	SR_TempDeviationToHighB[5](SET1:=mxAutoMode AND
((BottomMoldB.HeatingZone[5].FB_Temperature.EngTempOut > TopMoldB.HeatingZone[5].FB_Temperature.EngTempOut + 40.0)  OR 
( BottomMoldB.HeatingZone[5].FB_Temperature.EngTempOut < TopMoldB.HeatingZone[5].FB_Temperature.EngTempOut - 40.0)), RESET:=mxReset, Q1=>Errors.TempDeviationToHighB[5]);

	SR_TempDeviationToHighB[6](SET1:=mxAutoMode AND
((BottomMoldB.HeatingZone[6].FB_Temperature.EngTempOut > TopMoldB.HeatingZone[6].FB_Temperature.EngTempOut + 40.0)  OR 
( BottomMoldB.HeatingZone[6].FB_Temperature.EngTempOut < TopMoldB.HeatingZone[6].FB_Temperature.EngTempOut - 40.0)), RESET:=mxReset, Q1=>Errors.TempDeviationToHighB[6]);


(*Red hot safetyrule Regading heating Transfermold may not move down when bottommold A or B isn't hot enough*)
ASideNotWarm :=  ((BottomMoldA.HeatingZone[1].FB_Temperature.EngTempOut < MachParameters.MinTempAlowTransferToBot) AND MachParameters.BottomMoldA.HeatingZone[1].mxZoneActive) OR
				 ((BottomMoldA.HeatingZone[2].FB_Temperature.EngTempOut < MachParameters.MinTempAlowTransferToBot) AND MachParameters.BottomMoldA.HeatingZone[2].mxZoneActive) OR
				 ((BottomMoldA.HeatingZone[3].FB_Temperature.EngTempOut < MachParameters.MinTempAlowTransferToBot) AND MachParameters.BottomMoldA.HeatingZone[3].mxZoneActive) OR
				 ((BottomMoldA.HeatingZone[4].FB_Temperature.EngTempOut < MachParameters.MinTempAlowTransferToBot) AND MachParameters.BottomMoldA.HeatingZone[4].mxZoneActive) OR
				 ((BottomMoldA.HeatingZone[5].FB_Temperature.EngTempOut < MachParameters.MinTempAlowTransferToBot) AND MachParameters.BottomMoldA.HeatingZone[5].mxZoneActive) OR
				 ((BottomMoldA.HeatingZone[6].FB_Temperature.EngTempOut < MachParameters.MinTempAlowTransferToBot) AND MachParameters.BottomMoldA.HeatingZone[6].mxZoneActive);
		
BSideNotWarm :=  ((BottomMoldB.HeatingZone[1].FB_Temperature.EngTempOut < MachParameters.MinTempAlowTransferToBot) AND MachParameters.BottomMoldB.HeatingZone[1].mxZoneActive) OR
				 ((BottomMoldB.HeatingZone[2].FB_Temperature.EngTempOut < MachParameters.MinTempAlowTransferToBot) AND MachParameters.BottomMoldB.HeatingZone[2].mxZoneActive) OR
				 ((BottomMoldB.HeatingZone[3].FB_Temperature.EngTempOut < MachParameters.MinTempAlowTransferToBot) AND MachParameters.BottomMoldB.HeatingZone[3].mxZoneActive) OR
				 ((BottomMoldB.HeatingZone[4].FB_Temperature.EngTempOut < MachParameters.MinTempAlowTransferToBot) AND MachParameters.BottomMoldB.HeatingZone[4].mxZoneActive) OR
				 ((BottomMoldB.HeatingZone[5].FB_Temperature.EngTempOut < MachParameters.MinTempAlowTransferToBot) AND MachParameters.BottomMoldB.HeatingZone[5].mxZoneActive) OR
				 ((BottomMoldB.HeatingZone[6].FB_Temperature.EngTempOut < MachParameters.MinTempAlowTransferToBot) AND MachParameters.BottomMoldB.HeatingZone[6].mxZoneActive);
				
// FMEA (140 degree?)
SR_BotMoldAToCoolForTrMDown(SET1:=NOT mxCommisioningMode AND (BottomMoldA.mxCilIsIn AND ASideNotWarm AND TransferMold.mxCilIsMovingOut), Reset:=mxReset, Q1=>Errors.RH_BotMoldAToCoolForTrMDown);

SR_BotMoldBToCoolForTrMDown(Set1:= NOT mxCommisioningMode AND (BottomMoldB.mxCilIsIn AND BSideNotWarm AND TransferMold.mxCilIsMovingOut), reset:=mxReset, Q1=>Errors.RH_BotMoldBToCoolForTrMDown);
END_ACTION

ACTION Init:
(*StateChange (Transition)  Signalgeneration*)
mxInitTransitionState:=(miInitState<>miInitOldstate);
(*State text*)
sInitStateText:=sInitStateTextDef[miInitState];
(*Timeout Watchdog for Statemachine*)
mxInitTimeoutEnable:=NOT (miInitState=0)  AND NOT mxReset;

InitTimeout(IN:=mxInitTimeoutEnable  , PT:=tInitStateTimeouts[miInitState] );
InitTimeOutUpFlank(CLK:=InitTimeout.Q );
miInitOldstate:=miInitState;

(*Set Errorbit when Raising edge of Timeout has been detected*)
IF InitTimeOutUpFlank.Q THEN
	exInitTimeOut:=TRUE; 			(* 1 Timeout for the whole programcycle *)
END_IF

(*Function to reset the Statemachine*)
IF mxResetInitState THEN
	mxResetInitState:=FALSE;
	miInitState:=0;
	miInitOldstate:=miInitState;
	mxInitTransitionState:=FALSE;

	mxStartInit:= FALSE;
	mxStopInit:= FALSE;
	
	TopMoldA.mxResetInitState:= TRUE;
	TopMoldB.mxResetInitState:= TRUE;
	BottomMoldA.mxResetInitState:= TRUE;
	BottomMoldB.mxResetInitState:= TRUE;
	TransferMold.mxResetInitState:= TRUE;
	ProductForming.mxResetInitState:= TRUE;
	
END_IF

(*Definition State has Error*)
mxInitHasError:=FALSE;

(*Init State's*)
CASE miInitState OF
	0:
		IF mxStartInit THEN
			mxStartInit:= FALSE;
			mxInitialized:= FALSE;
			
			TransferMold.M_StartInit();
			ProductForming.M_StartInit();
			
			//HydraulicsMain.HydraulicPump.M_Start();
		
			miInitState:= 2;
		END_IF

	(* Init Transfermold / Product Forming*)
	2:
		IF mxStopInit THEN
			mxStopInit:= FALSE;
			
			miInitState:= 10;
		ELSIF TransferMold.mxInitialized AND ProductForming.mxInitialized THEN 
			IF MachParameters.EnableEamcSideA THEN
				TopMoldA.M_StartInit(); 

				miInitState:= 3;
			ELSIF MachParameters.EnableEamcSideB THEN
				TopMoldB.M_StartInit();

				miInitState:= 5; 
			END_IF
		END_IF

	(* Init topMold A *)
	3:
		IF mxStopInit THEN
			mxStopInit:= FALSE;
			
			miInitState:= 10;
		ELSIF TopMoldA.mxInitialized THEN
			BottomMoldA.M_StartInit();

			miInitState:= 4;
		END_IF

	(* Init BottomMold A *)	
	4:
		IF mxStopInit THEN
			mxStopInit:= FALSE;
			
			miInitState:= 10;
		ELSIF BottomMoldA.mxInitialized THEN
			IF MachParameters.EnableEamcSideB THEN
				TopMoldB.M_StartInit();

				miInitState:= 5; 
			ELSE
				//HydraulicsMain.M_SartInit();
				
				miInitState:= 7;
			END_IF
		END_IF

	(* Init topMold B *)
	5:
		IF mxStopInit THEN
			mxStopInit:= FALSE;
			
			miInitState:= 10;
		ELSIF TopMoldB.mxInitialized THEN
			BottomMoldB.M_StartInit();

			miInitState:= 6;
		END_IF

	(* Init BottomMold B *)	
	6:
		IF mxStopInit THEN
			mxStopInit:= FALSE;
			
			miInitState:= 10;
		ELSIF BottomMoldB.mxInitialized THEN
			//HydraulicsMain.M_SartInit();

			miInitState:= 7;
		END_IF

	(* Initialized *)
	7:
		mxInitialized:= TRUE;
		miInitState:= 0;
		
		//HydraulicsMain.HydraulicPump.M_Stop();
	(* Stop init *)
	10:
		mxInitialized:= FALSE;

		//HydraulicsMain.HydraulicPump.M_Stop();
		
		IF TopMoldA.mxInitBusy THEN TopMoldA.M_StopInit(); END_IF
		IF TopMoldB.mxInitBusy THEN TopMoldB.M_StopInit(); END_IF
		IF BottomMoldA.mxInitBusy THEN BottomMoldA.M_StopInit(); END_IF
		IF BottomMoldB.mxInitBusy THEN BottomMoldB.M_StopInit(); END_IF
		IF TransferMold.mxInitBusy THEN TransferMold.M_StopInit(); END_IF
		IF ProductForming.mxInitBusy THEN ProductForming.M_StopInit(); END_IF
		IF HydraulicsMain.mxInitbusy THEN HydraulicsMain.M_StopInit(); END_IF		

		miInitState:=11;
		
	(* Stop Init *)
	11:
		IF NOT TopMoldA.mxInitBusy AND NOT TopMoldB.mxInitBusy AND NOT BottomMoldA.mxInitBusy AND NOT BottomMoldB.mxInitBusy AND NOT TransferMold.mxInitBusy 
			AND NOT ProductForming.mxInitBusy AND NOT HydraulicsMain.mxInitbusy THEN	

			
			
			miInitState:= 0;
		END_IF
END_CASE

mxInitBusy:= miInitState<>0;
END_ACTION

METHOD M_StartCycle

IF (NOT mxCycleBusy AND mxInitialized) OR (mxInPause AND mxInitialized) THEN
	mxInPause:= FALSE;
	mxStartCycle:= TRUE;	
END_IF
END_METHOD

METHOD M_StartHydraulics : BOOL
HydraulicsMain.M_StartCycle();
END_METHOD

METHOD M_StartInit

IF NOT mxInitBusy THEN 
	mxStartInit:= TRUE; 
END_IF
END_METHOD

METHOD M_StopCycle

IF mxCycleBusy THEN
	mxStopCycle:= TRUE;	
	mxInPause:=TRUE;
END_IF
END_METHOD

METHOD M_StopCycleEmpty

IF mxCycleBusy THEN 
	mxStopCycleEmpty:= TRUE; 
END_IF
END_METHOD

METHOD M_StopDirect

IF mxCycleBusy THEN
	mxStopDirect:= TRUE;	
END_IF
END_METHOD

METHOD M_StopHydraulics
HydraulicsMain.M_StopCycleEmpty();
END_METHOD

METHOD M_StopInit

IF mxInitBusy THEN 
	mxStopInit:= TRUE; 
END_IF
END_METHOD

ACTION Objects:

TopMoldA(
	mxReset:= mxReset,
	mxEmergency:= mxEmergency[8],
	mxDoorsOpened:= mxEmergency[2] OR mxEmergency[3],
	mxAutoMode:= mxAutoMode,
	mxEnableHeating:= mxEnableHeating,	
	mxTakeOutIsMovingUp:= BottomMoldA.mxTakeoutIsMovingUp, 
	ActualPositionTransfermold:=Transfermold.ActualPosition,	
	RHSR_Blocked:= Errors.RH_ToMoldAIsMovingBoMoldANotInPos,
	MachParameters:= MachParameters.TopMoldA,
	ProdParameters:= ProdParameters.TopMoldA,
	Errors=> Errors.TopMoldA);

TopMoldB(
	mxReset:= mxReset,
	mxEmergency:= mxEmergency[8],
	mxDoorsOpened:=mxEmergency[3] OR mxEmergency[4],
	mxAutoMode:= mxAutoMode,
	mxEnableHeating:= mxEnableHeating,		
	mxTakeOutIsMovingUp:= BottomMoldB.mxTakeoutIsMovingUp, 
	ActualPositionTransfermold:=Transfermold.ActualPosition,
	RHSR_Blocked := Errors.RH_ToMoldBIsMovingBoMoldBNotInPos,
	MachParameters:= MachParameters.TopMoldB,
	ProdParameters:= ProdParameters.TopMoldB,
	Errors=> Errors.TopMoldB);
	
BottomMoldA(
	mxReset:= mxReset,
	mxEmergency:=mxEmergency[8],
	mxDoorsOpened:= mxEmergency[2] OR mxEmergency[3],
	mxAutoMode:= mxAutoMode,
	mxEnableHeating:= mxEnableHeating,		
	ActualPositionTransfermold:=Transfermold.ActualPosition,
	TransferPosA:= TransferMold.TransferPosA,
	TransferPosB:= TransferMold.TransferPosB,
	ContinueWithA:=ContinueWithA,
	ContinueWithB:=ContinueWithB,
	SgMoldsAreClosed := TopMoldA.SgTmIsDown,
	RHSR_Blocked := Errors.RH_BoMoldAIsMovingToMoldANotInPos OR Errors.RH_BoMoldAIsMovingTrMoldNotInPos OR Errors.RH_TaOutHorAIsMovingVertIsNotDown,
	mxGantryPickedUpProduct:= mxProductPickedUpGantry_A,
	MachParameters:= MachParameters.BottomMoldA,
	ProdParameters:= ProdParameters.BottomMoldA,
	SysParameters:= SysParameters.BottomMoldA,
	mxProductReadyAtTakeOut=> mxProductReadyAtTakeout_A,
	Errors=> Errors.BottomMoldA);

BottomMoldB(
	mxReset:= mxReset,
	mxEmergency:= mxEmergency[8],
	mxDoorsOpened:=mxEmergency[3] OR mxEmergency[4],
	mxAutoMode:= mxAutoMode,
	mxEnableHeating:= mxEnableHeating,
	ActualPositionTransfermold:=Transfermold.ActualPosition,
	TransferPosA:= TransferMold.TransferPosA,
	TransferPosB:= TransferMold.TransferPosB,
	ContinueWithA:=ContinueWithA,
	ContinueWithB:=ContinueWithB,
	SgMoldsAreClosed := TopMoldB.SgTmIsDown,	
	RHSR_Blocked := Errors.RH_BoMoldBIsMovingToMoldBNotInPos OR Errors.RH_BoMoldBIsMovingTrMoldNotInPos OR Errors.RH_TaOutHorBIsMovingVertIsNotDown,
	mxGantryPickedUpProduct:= mxProductPickedUpGantry_B,
	MachParameters:= MachParameters.BottomMoldB,
	ProdParameters:= ProdParameters.BottomMoldB,
	SysParameters:= SysParameters.BottomMoldB,
	mxProductReadyAtTakeOut=> mxProductReadyAtTakeout_B,
	Errors=> Errors.BottomMoldB);

TransferMold(
	mxReset:= mxReset,
	mxEmergency:= mxEmergency[2] OR mxEmergency[3] OR mxEmergency[4] OR mxEmergency[8],
	mxAutoMode:= mxAutoMode,
	mxStartVacuum:= ProductForming.mxStartTransferMoldVacuum,
	RHSR_Blocked:= Errors.RH_TrMoldIsMovingBoMoldANotInPos OR Errors.RH_TrMoldIsMovingBoMoldBNotInPos OR Errors.RH_TrMoldIsMovingSprayBNotInPos,
	MachParameters:= MachParameters.TransferMold,
	ProdParameters:= ProdParameters.TransferMold,
	Errors=> Errors.TransferMold);

	//TransferMold.mxCilIsMovingOut;
	
ProductForming( 
	mxReset:= mxReset,
	mxEmergency:= mxEmergency[2] OR mxEmergency[3] OR mxEmergency[4] OR mxEmergency[8],
	mxFirstCycle:= mxFirstCycle,
	mxAutoMode:= mxAutoMode,
	//sgTransferIsDown:= TransferMold.sgTrAtFormingPos,
	TransfermoldDownPosition:=TransferMold.DownPosition,
	TransfermoldMovingDown:=TransferMold.mxCilIsMovingOut,
	TransfermoldMovingUp:=Transfermold.mxCilIsMovingIn,
	ActualPositionTransfermold:=TransferMold.ActualPosition,
	RHSR_Blocked := FALSE,
	MachParameters:= MachParameters.ProductForming,
	SysParameters:= SysParameters.ProductForming,
	Errors=> Errors.ProductForming);

HydraulicsMain(
	mxReset:= mxReset,
	mxEmergency:=mxEmergency[8],	// All EM buttons.
	mxDoorOpened:=mxEmergency[2] OR mxEmergency[3] OR mxEmergency[4],	// Coresponding door zones have error.
	mxAutoMode:= mxAutoMode,
	mxHydraulicsReady => mxHydraulicsReady,
	PlcCycleTime:=PlcCycleTime,
	MachineParameters:= MachParameters.HydraulicsMain,
	Errors=>Errors.HydraulicMain);
END_ACTION

END_FUNCTION_BLOCK

// ---- POUs/InMoldDrying/TopMold/FB_TopMold.TcPOU
FUNCTION_BLOCK FB_TopMold
VAR CONSTANT
	sCycleStateTextDef: ARRAY[0..25]  OF STRING :=	
		['State 0: Wait for Start',
		'State 1: Wait for signal to start move down',
		'State 2: Move down',
		'State 3: Apply drying time',
		'State 4: Start drying',
		'State 5: Move up to open position with "open" speed',
		'State 6: Move up',
		'State 7: Wait until take out unit is up',
		'State 8: Await blowoff',
		'State 9: ',
		'State 10:',
		'State 11:',
		'State 12:',
		'State 13:',
		'State 14:',
		'State 15:',
		'State 16:',
		'State 17:',
		'State 18:',
		'State 19:',
		'State 20:[Pausing] Stop hydraulic movement',																
		'State 21:[Pausing] Move topmold to Up pause position',
		'State 22:[Paused] wait for start',
		'State 23:',
		'State 24:',
		'State 25:Stop direct state'];
	
	tCycleStateTimeouts: ARRAY[0..10] OF TIME := 
		[T#10S,T#10S,T#10S,T#10S,T#10S,T#10S,T#10S,T#10S,T#10S,T#10S,
		T#10S];

	sInitStateTextDef: ARRAY[0..10] OF STRING :=
		['State 0: Wait for Init Start',
		'State 1: Await pressure relief',
		'State 2: Move up',
		'State 3: Description Init State 3',
		'State 4: Description Init State 4',
		'State 5: Description Init State 5',
		'State 6: Description Init State 6',
		'State 7: Description Init State 7',
		'State 8: Description Init State 8',
		'State 9: Description Init State 9',
		'State 10: Stop init state'];

	tInitStateTimeouts: ARRAY[0..10] OF TIME := 
		[T#10S,T#10S,T#10S,T#10S,T#10S,T#10S,T#10S,T#10S,T#10S,T#10S
		,T#10S];
END_VAR

VAR_INPUT
	mxReset							: BOOL;	(*Reset Error*)
	mxEmergency						: BOOL;
	mxDoorsOpened					: BOOL;
	mxAutoMode						: BOOL; (* TRUE = Automode *)
	mxEmptyMachine					: BOOL;
	mxEnableHeating					: BOOL;

	mxResetCycleState				: BOOL;
	mxResetInitState				: BOOL;


	mxMoveUp						: BOOL; (* Drying finished or transfer ready with new product *)
	mxTakeOutIsMovingUp				: BOOL;
	ActualPositionTransfermold		: REAL;
	RHSR_Blocked 					: BOOL;
	
	(*Signals*)
	sgMoveDown						: BOOL; (* Signal from bottommold *)
	sgTakeOutUnitDown 				: BOOL;	(* Signal from bottommold *)
	sgSample						: BOOL; // Signals that a sample was taken out
	TopLateTime 					: REAL;
END_VAR
VAR_IN_OUT
	MachParameters					: ST_TopMoldMachPar;
	ProdParameters					: ST_TopMoldProdPar;

END_VAR
VAR_OUTPUT
(*Errors*)
	Errors							: ST_TopMoldErrors;
	mxErrorInit						: BOOL;		(* Error, stop immediately. Initialisation neccesary *)
	mxErrorStopinPos				: BOOL;		(* Error, stop in position. Only reset neccesary *)

(* State vars *)
	mxCycleBusy						: BOOL;
	mxInitBusy						: BOOL;
	
(* Vars *)
	mxInitialized					: BOOL;
	

	mxCilIsMovingIn					: BOOL;
	mxCilIsMovingOut				: BOOL;
	mxCilIsIn						: BOOL;
	mxCilIsOut						: BOOL;	
	ActualPosition					: REAL;
	
	MaxDryingSingleKO				: REAL;
	
(*Signals*)
	SgTmIsUp						: BOOL;	// Signals that the topmold is up
	SgTmIsDown						: BOOL; // Signals that the topmold is down

	SgElapsedDryingTime				: TIME;
	SgTotalDryingTime				: TIME;
	sgTopmoldBlowOffReady: BOOL;
END_VAR
VAR
(* State vars *)
	miCycleState					: INT :=0;
	miCycleOldstate					: INT :=0;
	mxCycleTransitionState			: BOOL := FALSE;
	sCycleStateText					: STRING;
	exCycleTimeOut					: BOOL;		(* Timeout for the whole programcycle *)
	CycleTimeout					: TON;
	CycleTimeOutUpFlank				: R_TRIG;
	mxCycleTimeoutEnable			: BOOL;
	CycleTime						: REAL;
	mxCycleHasError					: BOOL;
	miStopState						: INT;
	mxStartCycle					: BOOL;
	mxStopCycle						: BOOL;
	mxStopDirect					: BOOL;
	
	miInitState						: INT	:=0;
	miInitOldstate					: INT	:=0;
	mxInitTransitionState			: BOOL	:= FALSE;
	sInitStateText					: STRING;
	exInitTimeOut					: BOOL;		(* Timeout for the whole programcycle *)
	InitTimeout						: TON;
	InitTimeOutUpFlank				: R_TRIG;
	mxInitTimeoutEnable				: BOOL;
	InitTime						: REAL;
	mxInitHasError					: BOOL;
	mxStartInit						: BOOL;
	mxStopInit						: BOOL;
(* Objects *)
	HydraulicCilinder				: FB_HydraulicCilinderAnalog;
	Vacuum							: FB_MonoValveNoFdbck;
	BlowOff							: FB_MonoValveNoFdbck;
	HeatingZone						: ARRAY [1..6] OF FB_Heatingzone;
(* Vars *)
	T_DryingTime					: TON;
	T_BlowOffClosed					: TON;
	RT_TakeOutIsMovingUp			: R_TRIG;
	T_DryingMoldLock				: TON;
	T_VacuumTimeClosed				: TON;
	T_BlowOff						: TON;
	RT_EnableBlowOff				: R_TRIG;
	RT_EnableVacuum					: R_TRIG;
	RT_StartBlowOffClosed: R_TRIG;
	RT_StartVacuumClosed: R_TRIG;
	T_StartVacuumAfterDrying: TON;
	RT_StartVacuumAfterDrying: R_TRIG;
	TestTime: TIME := T#24500MS;
	T_PauseDelayedUp: TON;
	DryingTime: TIME;
	DryingElapsedTime: TIME;
	mxInPause: BOOL;

	T_SingleKO: TON;
	DryingSingleKO: REAL;
	T_TmNotOnBmPosTimeOut: TON;
	SR_TmDidNotReachBmPos: SR;
	RT_StartVacuumdEndDrying: R_TRIG;
END_VAR

Error();
Init();
Cycle();
Objects();

ActualPosition := HydraulicCilinder.ActPosition;

{region "Closed vacuum and blowoff HMI stuff"}
RT_EnableBlowOff(CLK:=MachParameters.EnableClosedBlowOff);
RT_EnableVacuum(CLK:=MachParameters.EnableClosedVacuum);

IF RT_EnableBlowOff.Q THEN
	MachParameters.EnableClosedVacuum := FALSE;
END_IF

IF RT_EnableVacuum.Q THEN
	MachParameters.EnableClosedBlowOff := FALSE;
END_IF
{endregion}

ACTION Cycle:
(*StateChange (Transition)  Signalgeneration*)
mxCycleTransitionState:=(miCycleState<>miCycleOldstate);
(*State text*)
sCycleStateText:=sCycleStateTextDef[miCycleState];
(*Timeout Watchdog for Statemachine*)
mxCycleTimeoutEnable:=NOT (miCycleState=0) AND NOT mxReset;

CycleTimeout(IN:=mxCycleTimeoutEnable  , PT:=tCycleStateTimeouts[miCycleState] );
CycleTimeOutUpFlank(CLK:=CycleTimeout.Q );
miCycleOldstate:=miCycleState;

(*Set Errorbit when Raising edge of Timeout has been detected*)
IF CycleTimeOutUpFlank.Q THEN
	exCycleTimeOut:=TRUE; 			(* 1 Timeout for the whole programcycle *)
END_IF

(*Function to reset the Statemachine*)
IF mxResetCycleState THEN
	mxResetCycleState:= FALSE;
	mxInitialized := FALSE;
		
	miCycleState:=0;
	miCycleOldstate:=miCycleState;
	mxCycleTransitionState:=FALSE;

	mxStartCycle:= FALSE;
	mxStopCycle:= FALSE;
	mxStopDirect:=FALSE;
	SgTmIsDown := FALSE;
	SgTmIsUp := FALSE;
	mxMoveUp := FALSE;
	sgMoveDown := FALSE;

	T_DryingTime.IN:= FALSE;
	T_DryingMoldLock.IN:= FALSE;
	T_VacuumTimeClosed.IN:= FALSE;
	T_BlowOffClosed.IN:= FALSE;
	T_BlowOff.IN:=FALSE;
	T_SingleKO.IN:= FALSE;
	DryingSingleKO := TIME_TO_REAL(T_SingleKO.ET);
	sgTopmoldBlowOffReady := FALSE;
	T_TmNotOnBmPosTimeOut.IN:=FALSE;	
	
	HydraulicCilinder.M_Stop();
END_IF

(*Definition State has Error*)
mxCycleHasError:=FALSE;

T_PauseDelayedUp(PT:=T#300MS);
T_BlowOff(IN:=, PT:=MachParameters.BlowOffToTakeOut);
T_DryingTime(IN:= , PT:= DryingTime);
SgElapsedDryingTime := T_DryingTime.ET;
SgTotalDryingTime := T_DryingTime.PT;
T_SingleKO(PT:=T#200S);
T_TmNotOnBmPosTimeOut(IN:=, PT:=T#5S);

{region "Vacuum / Blowoff while closed"}
	T_VacuumTimeClosed(IN:= , PT:= MachParameters.VacuumTimeClosed);
	T_BlowOffClosed(IN:= , PT:= MachParameters.BlowOffTimeClosed);	
	RT_StartBlowOffClosed(CLK:= MachParameters.EnableClosedBlowOff AND (miCycleState = 4));
	RT_StartVacuumClosed(CLK:=MachParameters.EnableClosedVacuum AND (miCycleState = 4));
	
	IF RT_StartBlowOffClosed.Q THEN 
		T_BlowOffClosed.IN := TRUE;
		BlowOff.M_On();
	ELSIF RT_StartVacuumClosed.Q THEN
		T_VacuumTimeClosed.IN := TRUE;
		Vacuum.M_On();
	END_IF
	
	IF T_BlowOffClosed.Q THEN 
		T_BlowOffClosed.IN := FALSE;
		BlowOff.M_Off(); 
	END_IF
	IF T_VacuumTimeClosed.Q THEN 
		T_VacuumTimeClosed.IN := FALSE;
		Vacuum.M_Off(); 
	END_IF
	
	RT_StartVacuumdEndDrying(CLK:=SgElapsedDryingTime > (SgTotalDryingTime - MachParameters.VacuumTimeEndDrying));
	IF RT_StartVacuumdEndDrying.Q THEN
		Vacuum.M_On();
	END_IF

{endregion}

{region "copy parameter set for pause position movement"}
	 MachParameters.PausePositionUpSlow := MachParameters.PositionUpSlow;	
	 MachParameters.PausePositionUpCreep := MachParameters.PositionUpCreep;	
{endregion}

(*Cycle State's*)
CASE miCycleState OF
	
	0:  // (P)  Wait for start
		IF mxStopCycle THEN
			mxStopCycle:= FALSE;
			miStopState:= miCycleState;
			miCycleState:= 20;
		ELSIF mxStartCycle THEN
			mxStartCycle:= FALSE;
			miCycleState:= 1;
		END_IF
	
	1:  // (P)  wait for move down
		HydraulicCilinder.M_Move(EndPosition:= MachParameters.PositionUpStop,  NormalSpeed:= MachParameters.SpeedUpNormal, 		// Keep topmold in its "up" position.
								SlowPosition:= MachParameters.PositionUpStop - MachParameters.PositionUpSlow, SlowSpeed:= MachParameters.SpeedUpSlow, 
								CreepPosition:=MachParameters.PositionUpStop - MachParameters.PositionUpCreep, CreepSpeed:=MachParameters.SpeedUpCreep);


		IF mxStopDirect THEN
			mxStopDirect:= FALSE;
			miCycleState:= 25;
		ELSIF mxStopCycle AND mxEmptyMachine THEN
			mxStopCycle:=False;
			mxEmptyMachine:= FALSE;
			HydraulicCilinder.M_Stop();
			miCycleState:= 0;
		ELSIF mxStopCycle THEN
			mxStopCycle:= FALSE;
			miStopState:= miCycleState;
			miCycleState:= 20;
		ELSIF sgMoveDown THEN
			T_SingleKO.IN:= FALSE;
			DryingSingleKO := TIME_TO_REAL(T_SingleKO.ET);
			sgTopmoldBlowOffReady := FALSE;
			sgMoveDown:= FALSE;
			mxMoveUp:= FALSE;
			SgTmIsUp:= FALSE;
			miCycleState:= 2;
		END_IF
	
	2:  // (NP) Move down. 
		T_TmNotOnBmPosTimeOut.IN:=TRUE;
		T_SingleKO.IN:= TRUE;
		IF mxStopDirect THEN
			mxStopDirect:= FALSE;
			miCycleState:= 25;(*Stop direct*)
		ELSIF MachParameters.UseNormalSpeedProfile AND NOT sgSample THEN
			IF HydraulicCilinder.M_Move(EndPosition:=ProdParameters.PositionDownStop, NormalSpeed:=MachParameters.SpeedDownNormal, 
										SlowPosition:=ProdParameters.PositionDownStop + Machparameters.PositionDownSlow, SlowSpeed:=MachParameters.SpeedDownNormal, 
										CreepPosition:=ProdParameters.PositionDownStop + Machparameters.PositionDownCreep, CreepSpeed:=MachParameters.SpeedDownNormal) OR T_TmNotOnBmPosTimeOut.Q THEN
			T_TmNotOnBmPosTimeOut.IN:=FALSE;
			sgSample := FALSE;
			miCycleState:= 3;
			END_IF
		ELSE											// go down with slow creep profile settings (also fist time after pause)
			IF HydraulicCilinder.M_Move(EndPosition:=ProdParameters.PositionDownStop, NormalSpeed:=MachParameters.SpeedDownNormal, 
										SlowPosition:=ProdParameters.PositionDownStop + Machparameters.PositionDownSlow, SlowSpeed:=MachParameters.SpeedDownSlow, 
										CreepPosition:=ProdParameters.PositionDownStop + Machparameters.PositionDownCreep, CreepSpeed:=MachParameters.SpeedDownCreep) OR T_TmNotOnBmPosTimeOut.Q THEN
			T_TmNotOnBmPosTimeOut.IN:=FALSE;
			sgSample := FALSE;
			miCycleState:= 3;
			END_IF
		END_IF
	
	3:  // (NP) Select HMI dryingtime
		IF mxStopDirect THEN
			mxStopDirect:= FALSE;
			miCycleState:= 25;(*Stop direct*)
		ELSIF TRUE  THEN
			Dryingtime := MachParameters.DryingTime;
			sgTmIsDown:= TRUE;
			sgTmIsUp:=FALSE;
			miCycleState:= 4;
		END_IF
	
	
	4:  // (P) start drying 
		T_DryingTime.IN:=TRUE;
		HydraulicCilinder.M_Press(Pressdown:=TRUE, PressSpeed:=MachParameters.PressSpeed, StoppingPressure:=MachParameters.PressStop);
		
		IF mxStopDirect THEN
			mxStopDirect:= FALSE;
			miCycleState:= 25;(*Stop direct*)
		ELSIF mxStopCycle THEN	
			DryingElapsedTime := T_DryingTime.ET;
			T_DryingTime.IN := FALSE;
			mxStopCycle:= FALSE;
			miStopState:= miCycleState;
			miCycleState:= 20;
		ELSIF T_DryingTime.Q THEN		// When dryingtime has finished, allways open up
			T_DryingTime.IN:= FALSE;
			Vacuum.M_On();
			miCycleState:= 5;
		END_IF
		
	5:  // (NP) Move up to "open" position with "slow" speed 
		IF mxStopDirect THEN
			mxStopDirect:= FALSE;
			miCycleState:= 25;
		//ELSIF HydraulicCilinder.M_Move(EndPosition:= ProdParameters.PositionDownOpen,  NormalSpeed:=MachParameters.SpeedOpening, 
		//								SlowPosition:= ProdParameters.PositionDownOpen, SlowSpeed:=MachParameters.SpeedOpening, 
		//								CreepPosition:=ProdParameters.PositionDownOpen, CreepSpeed:=MachParameters.SpeedOpening) THEN
		ELSIF TRUE THEN	
			miCycleState:= 6;
		END_IF
	
		
	6:  // (NP) Move up with product
		IF mxStopDirect THEN
			mxStopDirect:= FALSE;
			miCycleState:= 25;
		ELSIF HydraulicCilinder.M_OpenAndMove(EndPosition:= MachParameters.PositionUpStop,  NormalSpeed:= MachParameters.SpeedUpNormal, 
										SlowPosition:= MachParameters.PositionUpStop - MachParameters.PositionUpSlow, SlowSpeed:= MachParameters.SpeedUpSlow, 
										CreepPosition:=MachParameters.PositionUpStop - MachParameters.PositionUpCreep, CreepSpeed:=MachParameters.SpeedUpCreep,
										OpenPosition:= ProdParameters.PositionDownOpen,  OpenSpeed:=MachParameters.SpeedOpening) THEN
			SgTmIsUp:= TRUE;
			SgTmIsDown:= FALSE;
			mxMoveUp:= FALSE;
			miCycleState:= 7;
		END_IF
		
	7:  // (P) Wait until takeout is moving up
		IF mxStopDirect THEN
			mxStopDirect:= FALSE;
			miCycleState:= 25;(*Stop direct*)	
		ELSIF mxStopCycle THEN	
			mxStopCycle:= FALSE;
			miStopState:= miCycleState;
			miCycleState:= 20;
		ELSIF mxTakeOutIsMovingUp AND 
			HydraulicCilinder.M_Move(EndPosition:= MachParameters.PositionUpStop,  NormalSpeed:= MachParameters.SpeedUpNormal, 		// Keep topmold in its "up" position.
				SlowPosition:= MachParameters.PositionUpStop - MachParameters.PositionUpSlow, SlowSpeed:= MachParameters.SpeedUpSlow, 
				CreepPosition:=MachParameters.PositionUpStop - MachParameters.PositionUpCreep, CreepSpeed:=MachParameters.SpeedUpCreep) THEN
			Vacuum.M_Off();
			BlowOff.M_On();
			miCycleState:= 8;
		END_IF
		
	8:  // (P) Await Blowoff -> NP to P -> BaTeu 20190408 
		T_BlowOff.IN := TRUE;		
		IF mxStopDirect THEN
			mxStopDirect:= FALSE;
			miCycleState:= 25;(*Stop direct*)
		ELSIF mxStopCycle THEN	
			mxStopCycle:= FALSE;
			miStopState:= miCycleState;
			BlowOff.M_Off();
			miCycleState:= 20;
		ELSIF T_BlowOff.Q THEN			
			sgTopmoldBlowOffReady := TRUE;
			
			IF sgTakeOutUnitDown THEN
				BlowOff.M_Off();		
				T_BlowOff.IN := FALSE;
					
				miCycleState:= 1;
			END_IF
		END_IF
		
	20: //(NP) Pause step, stop all movement
		T_PauseDelayedUp.IN := TRUE;
		T_SingleKO.IN:= FALSE;
		DryingSingleKO := TIME_TO_REAL(T_SingleKO.ET);
		
		IF mxStopDirect THEN
			mxStopDirect:= FALSE;	
			miCycleState:= 25;
		ELSIF T_PauseDelayedUp.Q AND HydraulicCilinder.M_Stop() THEN		
			miCycleState:= 21;
		END_IF

	21: //(NP) Move up to pause position 
		IF mxStopDirect THEN
			mxStopDirect:= FALSE;
			miCycleState:= 25;
		ELSIF HydraulicCilinder.M_Move(EndPosition:=MachParameters.PausePositionUp, NormalSpeed:= MachParameters.SpeedUpSlow, 
											SlowPosition:=MachParameters.PausePositionUp - MachParameters.PausePositionUpSlow, SlowSpeed:=MachParameters.SpeedUpSlow,
											CreepPosition:=MachParameters.PausePositionUp - MachParameters.PausePositionUpCreep, CreepSpeed:=MachParameters.SpeedUpCreep) THEN
											
			HydraulicCilinder.M_Stop();
			miCycleState := 22;
		END_IF
		
	22: //(Paused) Await restart.
		IF mxStopDirect THEN
			mxStopDirect:= FALSE;
			miCycleState:= 25;
		ELSIF mxStartCycle THEN
			IF miStopState = 8 THEN	// if comming from state 8, restart blowoff.
				BlowOff.M_On();
			END_IF	
		
			IF miStopState = 4 THEN	// Re-calculate the remaining drying time and move down to drying pos.
				DryingTime := MachParameters.DryingTime - DryingElapsedTime;
					IF HydraulicCilinder.M_Move(EndPosition:=ProdParameters.PositionDownStop, NormalSpeed:=MachParameters.SpeedDownNormal, 		// Go down with slow creep profile
										SlowPosition:=ProdParameters.PositionDownStop + Machparameters.PositionDownSlow, SlowSpeed:=MachParameters.SpeedDownSlow, 
										CreepPosition:=ProdParameters.PositionDownStop + Machparameters.PositionDownCreep, CreepSpeed:=MachParameters.SpeedDownCreep) THEN
					mxStartCycle:= FALSE;
					miCycleState:= miStopState;
					END_IF
			ELSE					// Move to normal "up" position, and resume normal steps.
				IF HydraulicCilinder.M_Move(EndPosition:= MachParameters.PositionUpStop,  NormalSpeed:= MachParameters.SpeedUpSlow, 		
								SlowPosition:= MachParameters.PositionUpStop - MachParameters.PositionUpSlow, SlowSpeed:= MachParameters.SpeedUpSlow, 
								CreepPosition:=MachParameters.PositionUpStop - MachParameters.PositionUpCreep, CreepSpeed:=MachParameters.SpeedUpCreep) THEN	
					mxStartCycle:= FALSE;
					miCycleState:= miStopState;
				END_IF
			END_IF
		END_IF
		
	25: // Stop direct
		mxStartCycle:= FALSE;
		mxStopCycle:= FALSE;
		mxInitialized:= FALSE;

		T_DryingTime.IN:= FALSE;
		
		HydraulicCilinder.M_StopDirect();
		Vacuum.M_Off(); (* When product do not switch off *)
		BlowOff.M_Off();
		
		T_SingleKO.IN:= FALSE;
		DryingSingleKO := TIME_TO_REAL(T_SingleKO.ET);
		sgTopmoldBlowOffReady := FALSE;
		T_TmNotOnBmPosTimeOut.IN:=FALSE;		
		
		miCycleState:= 0;

END_CASE

mxCycleBusy:= miCycleState<>0 AND NOT (miCycleState=22);
mxInPause:=miCycleState=22;

IF (DryingSingleKO - TopLateTime) > 0 THEN
	MaxDryingSingleKO := (60000/(DryingSingleKO - TopLateTime));
END_IF
END_ACTION

ACTION Error:
SR_TmDidNotReachBmPos(SET1:=T_TmNotOnBmPosTimeOut.Q, RESET:= mxReset, Q1=>Errors.TmDidNotReachBmPosTimeOut);


(* ****************************************************************************** *)
mxErrorStopInPos:= Errors.TmDidNotReachBmPosTimeOut;
mxErrorInit:= HydraulicCilinder.mxErrorInit
			OR HeatingZone[1].mxErrorInit
			OR HeatingZone[2].mxErrorInit
			OR HeatingZone[3].mxErrorInit
			OR HeatingZone[4].mxErrorInit
			OR HeatingZone[5].mxErrorInit
			OR HEatingZone[6].mxErrorInit;
END_ACTION

ACTION Init:
(*StateChange (Transition)  Signalgeneration*)
mxInitTransitionState:=(miInitState<>miInitOldstate);
(*State text*)
sInitStateText:=sInitStateTextDef[miInitState];
(*Timeout Watchdog for Statemachine*)
mxInitTimeoutEnable:=NOT (miInitState=0)  AND NOT mxReset;

InitTimeout(IN:=mxInitTimeoutEnable  , PT:=tInitStateTimeouts[miInitState] );
InitTimeOutUpFlank(CLK:=InitTimeout.Q );
miInitOldstate:=miInitState;

(*Set Errorbit when Raising edge of Timeout has been detected*)
IF InitTimeOutUpFlank.Q THEN
	exInitTimeOut:=TRUE; 			(* 1 Timeout for the whole programcycle *)
END_IF

(*Function to reset the Statemachine*)
IF mxResetInitState THEN
	mxResetInitState:=FALSE;
	miInitState:=0;
	miInitOldstate:=miInitState;
	mxInitTransitionState:=FALSE;
	
	mxStartInit:= FALSE;
	mxStopInit:= FALSE;		
END_IF

(*Definition State has Error*)
mxInitHasError:=FALSE;

(*Init State's*)
CASE miInitState OF
	0:
		IF mxStartInit THEN
			mxStartInit:= FALSE;
			mxInitialized:=FALSE;
			
			Vacuum.M_Off();
			BlowOff.M_Off();

			miInitState:= 1;
		END_IF
		
	(* Move Up *)	
	1:
		IF mxStopInit THEN
			mxStopInit:= FALSE;

			miInitState:= 10;
		END_IF
			
		// Above Normal Position
		IF HydraulicCilinder.ActPosition > MachParameters.PositionUpStop THEN // Move down
			IF HydraulicCilinder.M_Move(EndPosition:=MachParameters.PositionUpStop, NormalSpeed:= MachParameters.InitSpeedDownNormal, 
											SlowPosition:=MachParameters.PositionUpStop + MachParameters.PositionUpSlow, SlowSpeed:=MachParameters.InitSpeeddownSlow, 
											CreepPosition:=MachParameters.PositionUpStop + MachParameters.PositionUpCreep,	CreepSpeed:=MachParameters.InitSpeedDownCreep ) THEN
			mxInitialized:= TRUE; (* Return val *)
			miInitState:= 0;	
			END_IF
		ELSE
		// Below normal position
			IF HydraulicCilinder.M_Move(EndPosition:=MachParameters.PositionUpStop, NormalSpeed:= MachParameters.InitSpeedUpNormal, 
											SlowPosition:=MachParameters.PositionUpStop - MachParameters.PositionUpSlow, SlowSpeed:=MachParameters.InitSpeedUpSlow, 
											CreepPosition:=MachParameters.PositionUpStop - MachParameters.PositionUpCreep,	CreepSpeed:=MachParameters.InitSpeedUpCreep ) THEN
			mxInitialized:= TRUE; (* Return val *)
			miInitState:= 0;	
			END_IF
		END_IF

	(* Stop Init *)
	10:
		HydraulicCilinder.M_Stop();

		mxStartInit:= FALSE;
		mxStopInit:= FALSE;
		mxInitialized:=FALSE;					

		miInitState:= 0;
END_CASE

mxInitBusy:= miInitState<>0;
END_ACTION

METHOD M_EmptyMachine

IF mxCycleBusy THEN
	mxEmptyMachine:= TRUE;	
END_IF
END_METHOD

METHOD M_StartCycle

IF NOT mxCycleBusy THEN
	mxStartCycle:= TRUE;	
	mxStopCycle := FALSE;
END_IF
END_METHOD

METHOD M_StartInit

IF NOT mxInitBusy THEN 
	mxStartInit:= TRUE; 
END_IF
END_METHOD

METHOD M_StopCycle
mxStopCycle:= TRUE;
END_METHOD

METHOD M_StopDirect

IF mxCycleBusy THEN
	mxStopDirect:= TRUE;	
END_IF
END_METHOD

METHOD M_StopInit

IF mxInitBusy THEN 
	mxStopInit:= TRUE; 
END_IF
END_METHOD

ACTION Objects:
(* Object Calls *)
HydraulicCilinder(
	mxReset:= mxReset, 
	mxEmergency:= mxEmergency OR mxDoorsOpened, 
	mxAutoMode:= mxAutoMode, 
	EndPositionIn:= MachParameters.PositionUpStop,
	EndPositionOut:= ProdParameters.PositionDownStop,
	OffsetPosition:= MachParameters.PositionOffsetZero,
	OffsetAlarmPosition:= MachParameters.PositionOffsetAlarm,
	PositionPhysicalMeasured:=MachParameters.PositionPhyscialMeasured,
	PositionPhysicalMeasuredOld:=MachParameters.PositionPhysicalMeasuredOld,
	PhysicalOffsetPos:=MachParameters.PhysicalOffsetPos,
	RHSR_Blocked:=RHSR_Blocked,
	mxCycleBusy:=mxCycleBusy,
	mxInitBusy:=mxInitBusy,
	mxIsMovingIn=> mxCilIsMovingIn, 
	mxIsMovingOut=> mxCilIsMovingOut, 
	ManSpeedCreepIn:=MachParameters.ManSpeedCreep,
	ManSpeedCreepOut:=MachParameters.ManSpeedCreep,
	ManSpeedSlowIn:=MachParameters.ManSpeedSlow,
	ManSpeedSlowOut:=MachParameters.ManSpeedSlow,
	ManSpeedIn:=MachParameters.ManSpeed,
	ManSpeedOut:=MachParameters.ManSpeed,
	mxIsIn=> mxCilIsIn, 
	mxIsOut=> mxCilIsOut,
	Errors=> Errors.Hydraulic);
	
Vacuum(
	mxReset:= mxReset, 
	mxEmergency:= mxEmergency OR mxDoorsOpened, 
	mxAutoMode:= mxAutoMode);
	
BlowOff(
	mxReset:= mxReset, 
	mxEmergency:= mxEmergency OR mxDoorsOpened, 
	mxAutoMode:= mxAutoMode);


HeatingZone[1](
	mxReset:= mxReset,
	mxEmergency:=mxEmergency OR mxDoorsOpened,
	mxDoorsOpened:=FALSE,
	mxEnableHeating:=mxEnableHeating,
	MachParameters:=MachParameters.HeatingZone[1],
	Errors=> Errors.HeatingZone[1]);	
	
HeatingZone[2](
	mxReset:= mxReset,
	mxEmergency:=mxEmergency OR mxDoorsOpened,
	mxDoorsOpened:=FALSE,
	mxEnableHeating:=mxEnableHeating,
	MachParameters:=MachParameters.HeatingZone[2],
	Errors=> Errors.HeatingZone[2]);

HeatingZone[3](
	mxReset:= mxReset,
	mxEmergency:=mxEmergency OR mxDoorsOpened,
	mxDoorsOpened:=FALSE,
	mxEnableHeating:=mxEnableHeating,
	MachParameters:=MachParameters.HeatingZone[3],
	Errors=> Errors.HeatingZone[3]);

HeatingZone[4](
	mxReset:= mxReset,
	mxEmergency:=mxEmergency OR mxDoorsOpened,
	mxDoorsOpened:=FALSE,
	mxEnableHeating:=mxEnableHeating,
	MachParameters:=MachParameters.HeatingZone[4],
	Errors=> Errors.HeatingZone[4]);

HeatingZone[5](
	mxReset:= mxReset,
	mxEmergency:=mxEmergency OR mxDoorsOpened,
	mxDoorsOpened:=FALSE,
	mxEnableHeating:=mxEnableHeating,
	MachParameters:=MachParameters.HeatingZone[5],
	Errors=> Errors.HeatingZone[5]);

HeatingZone[6](
	mxReset:= mxReset,
	mxEmergency:=mxEmergency OR mxDoorsOpened,
	mxDoorsOpened:=FALSE,
	mxEnableHeating:=mxEnableHeating,
	MachParameters:=MachParameters.HeatingZone[6],
	Errors=> Errors.HeatingZone[6]);
END_ACTION

END_FUNCTION_BLOCK

// ---- POUs/Standard/HydraulicCylinderAnalog/FB_HydraulicCilinderAnalog.TcPOU
FUNCTION_BLOCK FB_HydraulicCilinderAnalog

VAR_INPUT
	mxReset							: BOOL;	(*Reset Error*)
	mxEmergency						: BOOL;
	mxAutoMode						: BOOL; (* TRUE = Automode *)
	EndPositionIn					: REAL;
	EndPositionOut					: REAL;
	OffsetPosition					: REAL;
	OffsetAlarmPosition				: REAL;	
	PositionPhysicalMeasured		: REAL;	
	RHSR_Blocked					: BOOL; (*IF true, then movement of the cylinder is blocked by the red hot safetyrules.*)
	
	ManSpeedCreepIn					: REAL;
	ManSpeedCreepOut				: REAL;
	ManSpeedSlowIn					: REAL;
	ManSpeedSlowOut					: REAL;
	ManSpeedIn						: REAL;
	ManSpeedOut						: REAL;

END_VAR
VAR_OUTPUT
(*Errors*)
	Errors							: ST_HydraulicErrorsAnalog;
	mxErrorInit						: BOOL;		(* Error, stop immediately. Initialisation neccesary *)
	mxErrorStopinPos				: BOOL;		(* Error, stop in position. Only reset neccesary *)

(* State vars *)
	mxCycleBusy						: BOOL;
	mxInitBusy						: BOOL;
	
(* Vars *)
	mxInitialized					: BOOL;
	ActPosition						: REAL;
	ActMeasuredPosition				: REAL;
	mxSlowActive					: BOOL;
	mxIsMovingIn					: BOOL;
	mxIsMovingOut					: BOOL;
	mxIsIn							: BOOL;
	mxIsOut							: BOOL;
	mxMoveIn						: BOOL;
	mxMoveOut						: BOOL;
END_VAR
VAR
(* Testing new HMI alarms *)	
	_eventBase						: FB_TcEventBase;	
	_eventSourceName				: STRING;
	_translatedString				: STRING;
	_eventSourceInfo				: FB_TcSourceInfo;
	_asyncResult					: FB_AsyncStrResult;
	_initializeEvents				: BOOL := TRUE;
	_PositionError 					: FB_TcAlarm;
	_IsMovingWithoutActivationError	: FB_TcAlarm;
	_BallufError 					: FB_TcAlarm;

	RodSidePressure					: FB_AnalogIn4_20mA;
	BottomSidePressure				: FB_AnalogIn4_20mA;

	(* Objects *)
	HydraulicValve					: FB_AnalogOutMinus10_10V;
	HydraulicPos 					: FB_BalluffPosition;
	MachPar							: ST_HydraulicCilinderMachParAnalog;
	
	EndPosition						: REAL; (* Destination position *)
	SlowPosition					: REAL; (* Slow position *)

	FT_ValveInOff					: F_TRIG;
	FT_ValveOutOff					: F_TRIG;
	HydraulicStoredPosition			: REAL;
	
	ixEndSwitchA					AT %I* : BOOL;
	ixEndSwitchB					AT %I* : BOOL;
	ixMSPAReadyToOperate			AT %I* : BOOL;
	qxMSPAEnable					AT %Q* : BOOL;
	
	mxMoveReadyWithoutMoving		: BOOL;
	
	RT_Emergency: R_Trig;
	FT_AutoMode: F_TRIG;
	SafePosReached: BOOL;
	Mancreep: BOOL;
	ManCreepUp: BOOL;
	ManSlowUp: BOOL;
	ManUp: BOOL;
	ManCreepDown: BOOL;
	ManSlowDown: BOOL;
	ManDown: BOOL;
	SR_RodSidePressureTooHigh: SR;
	SR_BotSidePressureTooHigh: SR;
	T_EmergencyDelay: TON;
	RT_EmergencyDelay: R_TRIG;
	T_EnableDelayedOff: TOF;
	mxTestValue: REAL;
	FT_ValveToNeutralPos: F_trig;
	SR_SafePositionNotReached: SR;
END_VAR
VAR_IN_OUT
	PositionPhysicalMeasuredOld		: REAL;
	PhysicalOffsetPos				: REAL;
END_VAR

Error();
Objects();
Manual();

RT_Emergency(CLK:= mxEmergency);
FT_AutoMode(CLK:=mxAutoMode);

// Enable MSPA2
T_EnableDelayedOff(IN:= NOT mxEmergency, PT:=T#500MS);
qxMSPAEnable := T_EnableDelayedOff.Q; 

// Calculate correction on actual balluf position to a virtual "zero" position.
IF PositionPhysicalMeasured <> PositionPhysicalMeasuredOld THEN
	PhysicalOffsetPos := (HydraulicPos.Position- (OffsetPosition + PositionPhysicalMeasured));
END_IF

// Create a virtual zero position by substracting a calculated offset
ActPosition:= HydraulicPos.Position - PhysicalOffsetPos;
ActMeasuredPosition:= HydraulicPos.Position;

mxIsMovingIn:= HydraulicValve.EngInput > 0;
mxIsMovingOut:= HydraulicValve.EngInput < 0;

// Hysteresis + 2 to enlarge the RHSR window.
mxIsIn:= (ActPosition <= (EndPositionIn + (MachPar.Hysteresis + 2))) AND (ActPosition >= (EndPositionIn - (MachPar.Hysteresis + 2)));
mxIsOut:= (ActPosition <= (EndPositionOut + (MachPar.Hysteresis + 2))) AND (ActPosition >= (EndPositionOut - (MachPar.Hysteresis + 2)));

(*Overwrite previous value*)
PositionPhysicalMeasuredOld := PositionPhysicalMeasured;

// Close valves on emergency stop.
IF RT_Emergency.Q OR FT_AutoMode.Q THEN
	HydraulicValve.EngInput := 0;
END_IF

// From the TOP bosch -> If both feedback signals are high, the valve can be considered "safe" (base position reached
SafePosReached:= ixEndSwitchA AND ixEndSwitchB;

ACTION Error:
(* Initialize the alarms at the start *)
IF _initializeEvents THEN
	_initializeEvents := FALSE;
	_eventSourceName := _eventSourceInfo.sName;
	_PositionError.CreateEx(TC_Events.Kremer_Events.PositionError, TRUE, 0);
	_PositionError.ipArguments.Clear().AddString(_eventSourceName);
	_IsMovingWithoutActivationError.CreateEx(TC_Events.Kremer_Events.IsMovingWithoutActivation, TRUE, 0);
	_IsMovingWithoutActivationError.ipArguments.Clear().AddString(_eventSourceName);
	_BallufError.CreateEx(TC_Events.Kremer_Events.BallufError, TRUE, 0);
	
	_BallufError.RequestEventText(19, _translatedString, SIZEOF(_translatedString));
	_BallufError.RequestEventClassName(19, _translatedString, SIZEOF(_translatedString));
	
	(* _BallufError.ipArguments.Clear().AddString(_eventSourceName); *)
	
	
	F_GetEventText(19, _BallufError, _asyncResult);
	IF NOT _asyncResult.bBusy AND NOT _asyncResult.bError THEN 
		_asyncResult.GetString(_eventSourceName, SIZEOF(_eventSourceName));
		_BallufError.ipArguments.Clear().AddString(_eventSourceName);
	END_IF 
	
	(* _BallufError.SetJsonAttribute('{ "jsonKey":"jsonValue" }'); *)
END_IF

Errors.BallufError:= HydraulicPos.Error;
(* Raise the alarm *)
IF Errors.BallufError THEN
	_BallufError.Raise(0);
	(* _IsMovingWithoutActivationError.Raise(0);
	_PositionError.Raise(0); *)
ELSE
	IF _BallufError.eConfirmationState = 3 THEN (* If the alarm has been confirmed, clear it*)
		_BallufError.Clear(0, FALSE);
	END_IF
END_IF

// Check for a to high a pressure
SR_RodSidePressureTooHigh(SET1:=mxIsMovingIn AND (RodSidePressure.EngFilt > MachPar.MaxRodSidePressure),Reset:=mxReset,Q1=>Errors.RodSidePressureTooHigh);
SR_BotSidePressureTooHigh(SET1:=mxIsMovingOut AND (BottomSidePressure.EngFilt > MachPar.MaxBotSidePressure),Reset:=mxReset,Q1=>Errors.BotSidePressureTooHigh);	 

SR_SafePositionNotReached(SET1:=T_EmergencyDelay.Q AND NOT SafePosReached, reset:=mxReset, Q1=>Errors.SafePositionValveNotReached);

// Delay the emstop from the doors open, and wait checking on position.
T_EmergencyDelay(IN:=mxEmergency, PT:=T#500MS);
RT_EmergencyDelay(CLK:=T_EmergencyDelay.Q);

(* Als valve up/down uit gaat, positie opslaan en controleren of deze veranderd tov de act positie*)
IF RT_EmergencyDelay.Q THEN 
	HydraulicStoredPosition:= ActPosition; 
END_IF
IF mxReset THEN
	HydraulicStoredPosition:= ActPosition;
	Errors.IsMovingWithoutActivation:= FALSE;
ELSIF (T_EmergencyDelay.Q OR (HydraulicValve.EngInput = 0)) AND ((HydraulicStoredPosition > (ActPosition + 10)) OR (HydraulicStoredPosition < (ActPosition - 10))) THEN
	//Errors.IsMovingWithoutActivation:= TRUE;
END_IF

// Look into above alarm, this keeps triggering, probably due to not setting actual position in the right way

(***************************************************************************************)
mxErrorStopInPos:= Errors.PositionError OR Errors.IsMovingWithoutActivation OR Errors.BotSidePressureTooHigh OR Errors.RodSidePressureTooHigh;
mxErrorInit:= FALSE;
END_ACTION

METHOD M_Move : BOOL
VAR_INPUT
	EndPosition		: REAL; (* Destination position *)
	NormalSpeed		: REAL;
	
	SlowPosition	: REAL; (* Slow position *)
	SlowSpeed		: REAL;
		
	CreepPosition 	: REAL;	(*CreepSpeed.*)
	CreepSpeed		: REAL;
	
END_VAR
VAR_OUTPUT
END_VAR
VAR


	mxMoveINReady: BOOL;
	mxMoveOutReady: BOOL;
	ActSpeed : real;

	End_Position: REAL;
	Slow_Position: REAL;
	Creep_Position: REAL;
	Normal_Speed: REAL;
	Slow_Speed: REAL;
	Creep_Speed: REAL;
END_VAR
mxMoveReadyWithoutMoving := FALSE;

//Check current position of the rod, and check where to go and detemine direction
IF ActPosition > (EndPosition + MachPar.Hysteresis) THEN		// Move up (Positive)
	(*Set movement direction bit.*)
	mxMoveIn:= FALSE;
	mxMoveOut:= TRUE;
	ActSpeed:= NormalSpeed;
ELSIF ActPosition < (EndPosition - MachPar.Hysteresis) THEN 	// Move Down (Negative)
	(*Set movement direction bit.*)
	mxMoveIn:= TRUE;
	mxMoveOut:= FALSE;
	ActSpeed:= NormalSpeed;
ELSE																			// Don't move at all (allready on pos).
	mxMoveIn:= FALSE;
	mxMoveOut:= FALSE;
	mxMoveReadyWithoutMoving := TRUE;
END_IF

// Check at which speed the movement needs to be done.
IF (NOT mxMoveIn AND NOT mxMoveOut) THEN	// No movement.
	ActSpeed:= 0;
ELSIF (mxMoveIn AND (ActPosition > CreepPosition)) OR (mxMoveOut AND (ActPosition < CreepPosition)) THEN 	//Creep speed.
	ActSpeed:= CreepSpeed;
ELSIF (mxMoveIn AND (ActPosition > SlowPosition)) OR (mxMoveOut AND (ActPosition < SlowPosition)) THEN 		//Slow speed.
	ActSpeed:= SlowSpeed;
ELSIF (mxMoveIn OR mxMoveOut) THEN	// Normal speed if nothing else is selected.
	ActSpeed:= NormalSpeed;
END_IF

// Set actual output on valve.
IF mxMoveOut THEN ActSpeed := Actspeed *-1; END_IF
HydraulicValve.EngInput := ActSpeed;

// Check if the movement is ready.
mxMoveInReady := (mxMoveIn AND ((ActPosition >= (EndPosition - MachPar.Hysteresis)) AND 
				(ActPosition <= (EndPosition + MachPar.Hysteresis))));
mxMoveOutReady := (mxMoveOut AND ((ActPosition >= (EndPosition - MachPar.Hysteresis)) AND 
				(ActPosition <= (EndPosition + MachPar.Hysteresis))));	

// reset directional bits to zero when leaving this method.
IF mxMoveInReady OR mxMoveOutReady OR mxMoveReadyWithoutMoving THEN
	mxMoveIn:= FALSE;
	MxMoveOut:= FALSE;
END_IF

// Signal the method has finished to the caller of the method.
M_MOVE := mxMoveInReady OR mxMoveOutReady OR mxMoveReadyWithoutMoving;
END_METHOD

METHOD M_Press : BOOL
VAR_INPUT
	PressDown		 	: BOOL; // Determines if press needs to be done moving down 
	PressSpeed			: REAL;	// Flow at which the pressing occures
	StoppingPressure	: REAL;	// Pressure at which the pressing stops
END_VAR
VAR_OUTPUT
END_VAR
VAR
	PressingDone		: Bool;
END_VAR
IF PressDown THEN	// PressDown
	IF (BottomSidePressure.EngFilt < StoppingPressure - 15) THEN
		HydraulicValve.EngInput := PressSpeed * -1;
	END_IF
		
	IF (BottomSidePressure.EngFilt > StoppingPressure) THEN 
		HydraulicValve.EngInput := 0;			
		M_Press := TRUE;	// Signal the method is done.
	END_IF 	
ELSE				// PressUp
	IF (RodSidePressure.EngFilt < StoppingPressure) THEN
		HydraulicValve.EngInput := PressSpeed;
	ELSE
		HydraulicValve.EngInput := 0;	
		M_Press := TRUE;	// Signal the method is done.
	END_IF 
END_IF
END_METHOD

METHOD M_Stop : BOOL;
mxMoveIn := FALSE;
mxMoveOut := FALSE;

HydraulicValve.EngInput := 0.0;

M_Stop:= TRUE;
END_METHOD

METHOD M_StopDirect
HydraulicValve.EngInput := 0.0;
END_METHOD

ACTION Manual:
IF ManCreepUp THEN
	HydraulicValve.EngInput := ManSpeedCreepIn;
ELSIF ManSlowUp THEN
	HydraulicValve.EngInput := ManSpeedSlowIn;
ELSIF ManUp THEN
	HydraulicValve.EngInput := ManSpeedIn;
ELSIF ManCreepDown THEN
	HydraulicValve.EngInput := ManSpeedCreepOut * -1;
ELSIF ManSlowDown THEN
	HydraulicValve.EngInput := ManSpeedslowOut * -1;
ELSIF ManDown THEN											// Somebody is seriously wounded. ^_^
	HydraulicValve.EngInput := ManSpeedOut * -1;
END_IF

FT_ValveToNeutralPos(CLK:=ManCreepUp OR ManSlowUp OR ManUp OR ManCreepDown OR ManSlowDown OR ManDown);

// When Automode is disabled, set the valve back to neutral position.
IF FT_AutoMode.Q OR Ft_ValveToNeutralPos.Q THEN
	HydraulicValve.EngInput := 0.0;
END_IF
END_ACTION

ACTION Objects:
(* Objects Call *)
BottomSidePressure(
	EngLowLimit:=0, 
	EngUpperLimit:=315, 
	maOut=> , 
	EngUnits=> , 
	EngFilt=> , 
	OverRange=> , 
	UnderRange=> );

RodSidePressure(
	EngLowLimit:=0, 
	EngUpperLimit:=315, 
	maOut=> , 
	EngUnits=> , 
	EngFilt=> ,
	OverRange=> ,
	UnderRange=> );
	
HydraulicValve( 
	EngMin:= -100,
	EngMax:= 100,
	RHSR_Blocked:= RHSR_Blocked,
	VOut=> , 
	RawOut=> );
	
HydraulicPos();
END_ACTION

END_FUNCTION_BLOCK

// ---- POUs/Standard/Analog/FB_AnalogIn4_20mA.TcPOU
FUNCTION_BLOCK FB_AnalogIn4_20mA
VAR_INPUT
	EngLowLimit				: REAL; (*Low limit*)
	EngUpperLimit 			: REAL; (*Upper limit*)
END_VAR
VAR_OUTPUT
	maOut 					: REAL;
	EngUnits 				: REAL; (*Output in engineering units*)
	EngFilt 				: REAL; (*Gefilterde output*)
	OverRange				: BOOL;
	UnderRange				: BOOL;
END_VAR
VAR
	RawInput				AT%I*	:INT;
	Status					AT%I*	:BYTE;
	Buffer					: ARRAY [1..50] OF REAL;
	X						: INT;
	Filton 					: BOOL:=TRUE;
	FilterSize				: INT:=10;

END_VAR

OverRange:=FALSE;
UnderRange:=FALSE;

IF Status<=0 THEN
  mAOut:=(20.0-4.0)/32767*RawInput+4;
  Engunits:=(EngUpperLimit-EngLowLimit)/32767*RawInput+EngLowLimit;
ELSE
 mAOut:=Engunits:=(EngUpperLimit-EngLowLimit)/32767*RawInput+EngLowLimit;
 Engunits:= Engunits:=(EngUpperLimit-EngLowLimit)/32767*RawInput+EngLowLimit;
 OverRange:=(2 AND Status)>0;
 UnderRange:=(1 AND Status)>0;
  IF ((NOT OverRange) AND (NOT UnderRange)) THEN
       OverRange:=TRUE;
	UnderRange:=TRUE;
  END_IF;
END_IF;

(*Wanneer Filter Geactiveerd dan loop filter waarden door*)
IF Filton THEN
	Engfilt:=0;
   (*Schuif waarden door in buffer*)
	FOR x:=1 TO FilterSize-1 DO
          	Buffer[x]:=Buffer[x+1];
		EngFilt:=EngFilt+Buffer[x];
	END_FOR
   Buffer[FilterSize]:=Engunits;
   (*Gefilterde output is gemiddelde laatste x waarden*)
   EngFilt:=(Engfilt+Engunits)/FilterSize;
END_IF

END_FUNCTION_BLOCK

// ---- POUs/Standard/Analog/FB_AnalogOutMinus10_10V.TcPOU
FUNCTION_BLOCK FB_AnalogOutMinus10_10V
VAR_INPUT
	EngInput			: REAL;
	EngMin			: REAL; (* Lower limit Engineering units*)
	EngMax 			: REAL; (* Upper limit Engineering units*)
	RHSR_Blocked 	: BOOL; // Indicates whether this part is free to move (operate).
END_VAR
VAR_OUTPUT
	VOut 			: REAL;
	RawOut 			: INT;
END_VAR
VAR
	Input			: REAL;

	qwOutput			AT %Q*: INT;
END_VAR

Input:= LIMIT(EngMin, EngInput, EngMax);

IF EngMin <> 0 AND Engmax <> 0 THEN (* Check if min max <> 0, prevent division by zero *)
	IF Input > 0 THEN (* + 10 Volt part *)
		RawOut:= REAL_TO_INT(32767.0 * (Input / EngMax));
		VOut:= 10 * (RawOut/32767.0);
	ELSIF Input < 0 THEN (* - 10 Volt part *)
		RawOut:= -1 * REAL_TO_INT(32767.0 * (Input/EngMin));
		VOut:= 10 * (RawOut/32767.0);
	ELSE
		RawOut:=0;
		VOut:= 0;
	END_IF
END_IF

IF NOT RHSR_Blocked THEN
	qwOutput:= RawOut;
ELSE
	qwOutput := 0;
END_IF

END_FUNCTION_BLOCK

// ---- POUs/Standard/Balluff/FB_BalluffPosition.TcPOU
FUNCTION_BLOCK FB_BalluffPosition
VAR_INPUT
END_VAR
VAR_OUTPUT
	Error	: BOOL;
	Position: REAL;
	Temperature	: REAL;
END_VAR
VAR
	Magnet AT %I* : ST_BalluffMagnet;
END_VAR

Error:= (Magnet.PosAboveWorkAreaHighLimit<>0) OR (Magnet.PosBelowWorkAreaLowLimit<>0) OR (Magnet.PosMarkerFailure<>0);
Position:= DINT_TO_REAL(Magnet.Position)/1000.0;

END_FUNCTION_BLOCK

// ---- POUs/Standard/Valves/FB_MonoValveNoFdbck.TcPOU
FUNCTION_BLOCK FB_MonoValveNoFdbck
VAR_INPUT
	mxReset						: BOOL;	(*Reset Error*)
	mxEmergency					: BOOL;
	mxAutoMode					: BOOL; (* TRUE = Automode *)
	RHSR_Blocked				: BOOL := FALSE;
	SlowValveIsInverted			: BOOL := FALSE;
	mxDisableManualAutoTrigger	: BOOL := FALSE;
END_VAR
VAR_OUTPUT
	mxIsOn						: BOOL;
END_VAR
VAR
	Q	 						AT %Q*: BOOL;
	
	mxHMI_On					: BOOL;
	RT_HMI_On					: R_TRIG;
	RT_HMI_Off					: R_TRIG;
	RT_AutoMode					: R_TRIG;
	FT_AutoMode					: F_TRIG;
END_VAR

RT_HMI_On(CLK:=mxHMI_On);
RT_HMI_Off(CLK:=NOT mxHMI_On);
RT_AutoMode(CLK:= mxAutoMode);
FT_AutoMode(CLK:= mxAutoMode);

IF (RT_HMI_On.Q AND NOT mxAutoMode) AND NOT RHSR_Blocked THEN M_On(); END_IF
IF ((RT_HMI_Off.Q AND NOT mxAutoMode) OR ((RT_AutoMode.Q OR FT_AutoMode.Q) AND NOT mxDisableManualAutoTrigger)) OR RHSR_Blocked THEN M_Off(); END_IF

IF NOT SlowValveIsInverted THEN
mxIsOn:= Q; 
ELSE
mxIsOn:= NOT Q;
END_IF

METHOD PUBLIC M_Off : BOOL

VAR_INPUT
END_VAR
Q:=SlowValveIsInverted;

(* Return Value *)
M_Off:= TRUE;
END_METHOD

METHOD PUBLIC M_On : BOOL
VAR_INPUT
END_VAR
Q:=NOT SlowValveIsInverted;

(* Return Value *)
M_On:= TRUE;
END_METHOD

END_FUNCTION_BLOCK

// ---- POUs/Standard/HeatingZone/FB_HeatingZone.TcPOU
FUNCTION_BLOCK PUBLIC FB_HeatingZone
VAR_INPUT
	mxEnableHeating 				: BOOL;
	mxReset							: BOOL;
	mxEmergency						: BOOL;
	mxDoorsOpened					: BOOL;
END_VAR
VAR_OUTPUT
	mxErrorInit						: BOOL;
	mxErrorStopInPos				: BOOL;
	Errors							: ST_HeatingZoneErrors;
END_VAR
VAR

	qxPWMOut1 AT%Q*					: BOOL;
	qxPWMOut2 AT%Q*					: BOOL;
	qxPWMOut3 AT%Q*					: BOOL;
	ixThermal AT%I*					: BOOL;
	
	FT_EnableHeating				:F_Trig;	

	FB_Heating_Controller			: FB_PIDCtrl;
	FB_PID							: FB_PID_CP;
	FB_PWM							: FB_CTRL_PWM_OUT;
	FB_Temperature					: FB_AnalogInPT100;
	RT_EmStop						: R_TRIG;
	FT_EmStop						: F_TRIG;
	ControlMode						: E_CTRL_MODE;
	RT_ActivateHeating				: R_TRIG;
	RT_TempError					: R_TRIG;
	
	T_TempBelowSetpoint				: TON;
	SR_TempBelowSetpoint			: SR;
	T_TempAboveSetpoint				: TON;
	SR_TempAboveSetpoint			: SR;
	T_TimeInAutomode				: TON;

	T_HeatingStarted				: TON;

	SR_PT100_Loose					: SR;
	SR_PT100_WireBreakActive		: SR;
	SR_PT100_HasWrongPosition		: SR;
	SR_PT100_NotInserted			: SR;
	SR_PT100_ConnectorNotConnected	: SR;
	SR_PT100_ResistorFound	: SR;
	
	T_PT100_CheckTemperatures		: TON;
	mxIncreasedTemperatureNonActive	: BOOL;
	mxNoIncreaseTemperatureActive	: BOOL;
	OldTemperature					: REAL;
	
	T_PT100_HasWrongPosition		: Ton;
	FT_ActivateHeating: F_TRIG;
	SR_PT100_EnabledZoneWithoutProperPt100: SR;
	SR_TemperatureWayTooHigh: SR;
	
	Setpoint 			 	: REAL;
	TemperatureDifference	: REAL;
	SetpointStep		 	: REAL;
	ActStepNr            	: INT;
	ActTempMemory 			: REAL;
	PIDsetpoint				: REAL;
	mxSetpointReached		: BOOL;
	T_TempAtSetpointDelayNextStep	: TON;
	RT_StartHeatingInSteps			: R_TRIG;
	HeatingInSteps					: BOOL;
	RT_StopHeatingInSteps: R_TRIG;
	RT_DoorOpened: R_TRIG;
	FT_DoorOpened: F_TRIG;
	RT_HeatingPIDON: R_TRIG;
	FT_HeatingPIDON: F_TRIG;
	RT_SetPointChanged: R_TRIG;
	OldSetpoint: REAL; 
	SR_TemperatureTooHighWarning: SR;
END_VAR
VAR_IN_OUT
	MachParameters					: ST_HeatingZone;
END_VAR

DetermineSetpoint();
Error();
Objects();

RT_ActivateHeating(CLK:=MachParameters.mxZoneActive);
T_HeatingStarted(IN:=, PT:=T#10M);

RT_HeatingPIDON(CLK:=FB_Heating_Controller.PID_ON);
FT_HeatingPIDON(CLK:=FB_Heating_Controller.PID_ON);

FB_Heating_Controller.PID_ON := mxEnableHeating AND MachParameters.mxZoneActive AND NOT mxEmergency AND NOT FB_Temperature.Error;

// Start heating "started" timer when heating switches on
IF RT_HeatingPIDON.Q THEN
	T_HeatingStarted.IN := TRUE;
END_IF

IF NOT FB_Heating_Controller.PID_ON THEN
	T_HeatingStarted.IN :=FALSE;
END_IF

// Autoreset the PWM controller when a error occures
IF FB_PWM.bError AND (ControlMode = eCTRL_MODE_ACTIVE) THEN
	Controlmode := eCTRL_MODE_RESET;
ELSE
	ControlMode := eCTRL_MODE_ACTIVE;
END_IF

OldSetpoint := MachParameters.PIDTempZone.SP_AUTO;

ACTION DetermineSetpoint:
// because of enormous overshoots, the setpoint of the PID is scaled up during startup
// and cut into smaller heating steps. For example when a 180 degree setpoint is set in the HMI
// And the number of warmingsteps is set to 10. The PID first gets a setpoint of: 180/10 * 1
// When the setpoint is reached the timer "SetpointReached" starts counting. When this timer
// is elapsed the next set is set into the PID -> 180/10 * 2.


RT_StartHeatingInSteps(CLK:=(FB_Heating_Controller.PV_EXT < MachParameters.LowLimitSP) AND RT_HeatingPIDON.Q);
RT_StopHeatingInSteps(CLK:=FT_HeatingPIDON.Q, Q=>);
T_TempAtSetpointDelayNextStep(IN:=mxSetpointReached, PT:=MachParameters.WaitTimeAfterStepReached);

// Interupt/stop heating in steps.
IF RT_StopHeatingInSteps.Q THEN HeatingInSteps:= FALSE; END_IF

//do this once when starting heating, determine setpoints.
IF RT_StartHeatingInSteps.q THEN
	HeatingInSteps := TRUE;
	
	TemperatureDifference := MachParameters.PIDTempZone.SP_AUTO_TOTAL - FB_Heating_Controller.PV_EXT;		// 160 = 180 - 20
	SetpointStep := TemperatureDifference / MachParameters.nrOfSteps;								// 16  = 160 / 10
	ActStepNr := 1;
	ActTempMemory := FB_Heating_Controller.PV_EXT;
	MachParameters.PIDTempZone.SP_AUTO := (ActStepNr * SetpointStep) + ActTempMemory;										// 1 * 16.0 + 20 =36.0 degree
END_IF

// When heating in steps is active the following code is active
IF HeatingInSteps THEN
		
	IF NOT mxSetpointReached AND (FB_Heating_Controller.PV_EXT >= MachParameters.PIDTempZone.SP_AUTO) THEN mxSetpointReached := TRUE; END_IF	
	
	IF T_TempAtSetpointDelayNextStep.q THEN
		
		mxSetpointReached := FALSE;
		
		IF ActStepNr < MachParameters.nrOfSteps THEN
			ActStepNr := ActStepNr + 1;
			MachParameters.PIDTempZone.SP_AUTO := (ActStepNr * SetpointStep) + ActTempMemory;			// 1 * 16.0 + 20 =36.0 degree
		ELSE
			ActStepNr := 1;
			HeatingInSteps := FALSE;
		END_IF;
			
	END_IF;
ELSE
	MachParameters.PIDTempZone.SP_AUTO := MachParameters.PIDTempZone.SP_AUTO_TOTAL;
END_IF;
END_ACTION

ACTION Error:
// FMEA errors .. //

//1 PT100 loose
SR_PT100_Loose(SET1:=SR_PT100_WireBreakActive.Q1 OR T_PT100_HasWrongPosition.Q OR SR_PT100_NotInserted.Q1, RESET:=mxReset, Q1=> );

//2 Wire break alarm (from terminal).
SR_PT100_WireBreakActive(Set1:= FB_Temperature.Wirebreak, Reset:=mxReset);

//3 check heating element zone, check if there is no difference in temperature over a x time while element is active
SR_PT100_HasWrongPosition(SET1:=NOT mxEmergency AND mxEnableHeating AND MachParameters.mxZoneActive AND mxNoIncreaseTemperatureActive  
AND (FB_Temperature.EngTempOut < (MachParameters.PIDTempZone.SP_AUTO - 40.0))  , Reset:=mxReset);

//4 check heating element zone, check if there is a difference in temperature over a x time while element is not
SR_PT100_NotInserted(SET1:=((NOT MachParameters.mxZoneActive) AND mxIncreasedTemperatureNonActive AND NOT T_HeatingStarted.Q), Reset:=mxReset); // testen!

// Other errors.. //
SR_PT100_EnabledZoneWithoutProperPt100(SET1:=(FB_Temperature.EngTempOut < 5.0) AND RT_ActivateHeating.Q, RESET:=mxReset );

IF (FB_Temperature.EngTempOut < 5.0) OR Errors.PT100_TemperatureAboveMaximum THEN
	MachParameters.mxZoneActive := FALSE;
END_IF

// Connector pt100 not connected: 100 ohm missing / pt100 , open loop.
SR_PT100_ConnectorNotConnected(SET1:=(FB_Temperature.EngTempOut > 750) , RESET:=mxReset);

// Is a warning now only, only alarm message in the HMI 
SR_TempBelowSetpoint(SET1:=T_TempBelowSetpoint.Q , RESET:= mxReset);
SR_TempAboveSetpoint(SET1:=T_TempAboveSetpoint.Q , RESET:= mxReset);

// Alarming timers
T_TempBelowSetpoint(IN:= mxEnableHeating AND MachParameters.mxZoneActive AND (FB_Temperature.EngTempOut < (MachParameters.PIDTempZone.SP_AUTO -15)), PT:=T#1M);
T_TempAboveSetpoint(IN:= mxEnableHeating AND MachParameters.mxZoneActive AND (FB_Temperature.EngTempOut > (MachParameters.PIDTempZone.SP_AUTO +15)), PT:=T#1M);

// reset the timer of the change in temperature when the setpoint is changed on the HMI
RT_SetPointChanged(CLK:= OldSetpoint <> MachParameters.PIDTempZone.SP_AUTO);

T_PT100_CheckTemperatures(IN:= NOT T_PT100_CheckTemperatures.Q AND FB_Heating_Controller.PID_ON AND NOT RT_SetPointChanged.Q, PT:=MachParameters.TimeErrorCheckinterval);
IF T_PT100_CheckTemperatures.Q THEN
	mxNoIncreaseTemperatureActive := mxIncreasedTemperatureNonActive := FALSE;
	mxNoIncreaseTemperatureActive := mxEnableHeating AND NOT (FB_Temperature.EngTempOut > (OldTemperature + MachParameters.TempErrorRaise));
	mxIncreasedTemperatureNonActive := mxEnableHeating AND (FB_Temperature.EngTempOut > (OldTemperature + MachParameters.TempErrorRaise));
	OldTemperature := FB_Temperature.EngTempOut;
END_IF

IF NOT FB_Heating_Controller.PID_ON THEN mxNoIncreaseTemperatureActive := mxIncreasedTemperatureNonActive := FALSE; END_IF

SR_TemperatureWayTooHigh(SET1:=(FB_Temperature.EngTempOut > 250) AND (FB_Temperature.EngTempOut < 300.0), RESET:=mxReset);
SR_TemperatureTooHighWarning(SET1:=(FB_Temperature.EngTempOut > 230) AND (FB_Temperature.EngTempOut < 300.0), RESET:=mxReset);


Errors.Thermal:= NOT ixThermal;
Errors.PT100_Loose := SR_PT100_Loose.Q1;
Errors.PT100_WireBreak := SR_PT100_WireBreakActive.Q1;	
Errors.PT100_HasWrongPosition := SR_PT100_HasWrongPosition.Q1;
Errors.PT100_NotInserted := SR_PT100_NotInserted.Q1;
Errors.PT100_ConnectorNotConnected := SR_PT100_ConnectorNotConnected.Q1;
Errors.PT100_TemperatureAboveMaximum := SR_TemperatureWayTooHigh.Q1;
Errors.PT100_TemperatureTooHighWarn := SR_TemperatureTooHighWarning.Q1;
 
(**********************************************************************************************************)
mxErrorStopinPos:= FALSE; 
mxErrorInit:= errors.PT100_TemperatureAboveMaximum OR Errors.PT100_Loose;// OR Errors.PT100_ConnectorNotConnected;
END_ACTION

ACTION Objects:
FB_Temperature(
	EngTempOut=> , 
	Error=> );

FB_PID(
	Enable:= FB_Heating_Controller.PID_ON, 
	Reset:= NOT FB_Heating_Controller.PID_ON, 
	TskCycleTime:= T#10MS, 
	CtrlCycleTime:= T#20MS);
	
FB_Heating_Controller(
	PID:= FB_PID,
	PV_EXT:= FB_Temperature.EngTempOut, 
	Parameters:= MachParameters.PIDTempZone);

FB_PWM(
	fPwmInput:= FB_Heating_Controller.OUT_PID, 
	eMode:= Controlmode, 
	bPwmOutBitPos=> , 
	bPwmOutBitNeg=> , 
	eState=> , 
	eErrorId=> , 
	bError=> , 
	stParams:= MachParameters.PWM_Parameters);
	
MachParameters.PWM_Parameters.tTaskCycleTime := T#10MS;
	
	(*Generate output when this mold heating is enabled*)
qxPWMOut1:= qxPWMOut2:= qxPWMOut3:= FB_PWM.bPwmOutBitPos AND MachParameters.mxZoneActive;
END_ACTION

END_FUNCTION_BLOCK

// ---- POUs/Standard/HeatingZone/PID/FB_PIDCtrl.TcPOU
FUNCTION_BLOCK FB_PIDCtrl
VAR
	EU_Factor		: REAL; 			// Normalizing factor from EU-range (SP and PV) to 0-100 range 
	OUT_Factor		: REAL; 			// Normalizing factor from OUT-range to 0-100 range	
	LMN				: REAL;
	
	//PV_EXT			: REAL; 			// Process value 		
	PV_PID			: REAL;	
	PV_ACT			: REAL;
	
	HMI_SetpointBtn	: BOOL;
	HMI_AutoBtn		: BOOL;
	HMI_OutputBtn	: BOOL;
	
	
	//HMI_SetpointBtnState	: BOOL;
	//HMI_AutoBtnState		: BOOL;
	//HMI_OutputBtnState	: BOOL;

	RT_AutoBtnState: R_TRIG;
	RT_SetpointBtnState: R_TRIG;
	RT_OutBtnState: R_TRIG;

	FT_IL_ON: F_TRIG;
END_VAR
VAR_INPUT	
	PV_EXT			: REAL; 			// Process value 	
	PID_ON			: BOOL;				// switches the internal PID to operational mode or not.		
END_VAR
VAR_OUTPUT
	OUT_ACT			: REAL;
	OUT_PID			: REAL;
END_VAR
VAR_IN_OUT
	PID			: FB_PID_CP;			// Beckhoff PID controller															
//	SP_MAN		: REAL; 				// Setpoint manual				 					
//	OUT_MAN		: REAL; 				// Output manual 	
	Parameters: ST_PIDSettings;
END_VAR

RT_AutoBtnState(CLK:= HMI_AutoBtn);
RT_SetpointBtnState(CLK:= HMI_SetpointBtn);
RT_OutBtnState(CLK:= HMI_OutputBtn);

LMN		:= PID.LMN;
OUT_PID	:= PID.LMN;

(* Factor normering van EU range (SP en PV) naar 0-100 range		*)
IF (Parameters.EU_HLM - Parameters.EU_LLM) = 0 THEN
EU_Factor := 1.0;
ELSE
EU_Factor := 100.0 / (Parameters.EU_HLM - Parameters.EU_LLM);
END_IF


(* Setpoint					 										*)

//IF Status.Auto_Btn OR Status.M_Output_Btn
IF Parameters.AutoState OR Parameters.OutState THEN
	IF PID_ON
		THEN PID.SP_INT := (Parameters.SP_AUTO - Parameters.EU_LLM) * EU_Factor;
	END_IF

Parameters.SP_MAN := PID.SP / EU_Factor + Parameters.EU_LLM;
END_IF

IF Parameters.SetpointState THEN

	IF Parameters.SP_MAN < Parameters.SP_LLM_EXT
		THEN Parameters.SP_MAN := Parameters.SP_LLM_EXT;
	END_IF

	IF Parameters.SP_MAN > Parameters.SP_HLM_EXT
		THEN Parameters.SP_MAN := Parameters.SP_HLM_EXT;
	END_IF

PID.SP_INT := (Parameters.SP_MAN - Parameters.EU_LLM) * EU_Factor;
END_IF


Parameters.SP_PID := PID.SP / EU_Factor + Parameters.EU_LLM;

PID.SP_ROC := Parameters.SP_ROC_EXT * EU_Factor ;


PID.SP_LLM := (Parameters.SP_LLM_EXT - Parameters.EU_LLM) * EU_Factor;
PID.SP_HLM := (Parameters.SP_HLM_EXT - Parameters.EU_LLM) * EU_Factor;


(* Process Value					 										*)

PID.PV_IN := (PV_EXT - Parameters.EU_LLM) * EU_Factor;

IF Parameters.PV_TMLAG > 0.0
THEN
	PID.PV_TMLAG := Parameters.PV_TMLAG;
ELSE
	PID.PV_TMLAG := 0.0;
END_IF

(* Deadband					 										*)

IF Parameters.DEADBAND > 0.0
THEN
	PID.DEADBAND := Parameters.DEADBAND * EU_Factor;
ELSE
	PID.DEADBAND := 0.0;
END_IF

(* Linear reduction of I component in the innerwindow				*)
IF Parameters.fI_Innerwindow > 0.0
THEN
	PID.fI_InnerWindow := Parameters.fI_Innerwindow * EU_Factor;
ELSE
	PID.fI_InnerWindow := 0.0;
END_IF


(* Output															*)

(* Calculate Feedforward action	*)
Parameters.OUT_FF := Parameters.FF_GAIN * Parameters.FF_SIGNAL;

IF (Parameters.Out_MAX - Parameters.OUT_MIN) = 0 THEN
	OUT_Factor := 1.0;
ELSE
	OUT_Factor := 100.0 / (Parameters.Out_MAX - Parameters.OUT_MIN);
END_IF
IF NOT PID_ON
	AND NOT Parameters.SetpointState
	AND NOT Parameters.IL_ON
	AND NOT Parameters.OutState
THEN
PID.ManValue := 0.0;
END_IF

FT_IL_ON(CLK:=Parameters.IL_ON);

IF Parameters.IL_ON
	AND NOT Parameters.OutState
THEN
//PID.SP_INT := (PV_EXT - Parameters.EU_LLM) * EU_Factor;
PID.ManValue := Parameters.OUT_IL;
END_IF

IF FT_IL_ON.Q THEN
	PID.ManValue := Parameters.OUT_IL;
	PID.SP_INT := (PV_EXT - Parameters.EU_LLM) * EU_Factor;
END_IF


IF Parameters.OutState THEN
	IF Parameters.Out_MAN < Parameters.OUT_LLM_EXT THEN
		Parameters.Out_MAN := Parameters.OUT_LLM_EXT;
	END_IF

	IF Parameters.Out_MAN > Parameters.OUT_HLM_EXT THEN
		Parameters.Out_MAN := Parameters.OUT_HLM_EXT;
	END_IF
(* Fot bumpless transfer *)
PID.SP_INT := (PV_EXT - Parameters.EU_LLM) * EU_Factor;

PID.ManValue := (Parameters.Out_MAN - Parameters.OUT_FF - Parameters.OUT_MIN) * OUT_Factor;
END_IF

IF NOT Parameters.OutState THEN
Parameters.Out_MAN := (LMN + Parameters.OUT_FF)/ OUT_Factor + Parameters.OUT_MIN;
END_IF

IF NOT Parameters.RAUT_OP
	THEN LMN := 0.0;
END_IF



(* If Feedforward active, add feedforward to output and adjust boundaries of PID	*)
IF OUT_Factor >0 THEN
OUT_ACT := (LMN + Parameters.OUT_FF)/ OUT_Factor + Parameters.OUT_MIN;
END_IF
PID.LMN_LLM := (Parameters.OUT_LLM_EXT - Parameters.OUT_FF - Parameters.OUT_MIN) * OUT_Factor;
PID.LMN_HLM := (Parameters.OUT_HLM_EXT - Parameters.OUT_FF - Parameters.OUT_MIN) * OUT_Factor;

PID.LMN_ROC_UP := Parameters.Out_ROC_UP * OUT_Factor;
PID.LMN_ROC_DOWN := Parameters.Out_ROC_DOWN * OUT_Factor;

(* Output manual on					 										*)

PID.Man_On := Parameters.IL_ON OR Parameters.OutState;

(* Write PID parameters *)

PID.Kp 	:= 	Parameters.P;
PID.Tn 	:= 	Parameters.I;
PID.Tv 	:= 	Parameters.D;
PID.Td	:=  Parameters.Dtime;
PV_PID	:=	PID.PV;
PV_ACT	:=	(PID.PV/EU_Factor) + Parameters.EU_LLM;

PID.Invers	:= Parameters.INVERTED;

(* Status visualisation of limitation of output, ROC-out active *)
//Status.ROC_ACT	:= PID.FB_PID.bSync;

IF RT_AutoBtnState.Q THEN
	Parameters.AutoState := TRUE;	
	Parameters.SetpointState := FALSE;
	Parameters.OutState:=FALSE;
END_IF

IF RT_SetpointBtnState.Q THEN
	Parameters.AutoState := FALSE;	
	Parameters.SetpointState := TRUE;
	Parameters.OutState:=FALSE;
END_IF

IF RT_OutBtnState.Q THEN
	Parameters.AutoState := FALSE;	
	Parameters.SetpointState := FALSE;
	Parameters.OutState:=TRUE;
END_IF


// Low cutoff (make parameter.
IF Out_PID < Parameters.LowCutOff THEN
	OUT_PID := 0;
END_IF

IF OUT_PID > Parameters.HighCutOff AND Parameters.HighCutOff <> 0 THEN
	OUT_PID := Parameters.HighCutOff;
END_IF

END_FUNCTION_BLOCK

// ---- POUs/Standard/HeatingZone/PID/FB_PID_CP.TcPOU
FUNCTION_BLOCK FB_PID_CP
VAR
	FB_SP_ROC		: FB_PID_ROC;
	tTn				: TIME;
	tTv				: TIME;
	tTd				: TIME;
	SP				: REAL;
	PV				: REAL;
	fKp				: REAL;
	LMN_ROC_OUT		: REAL;
	SP_ROC_OUT		: REAL;
	PID_OUT			: REAL;
	FB_PID			: FB_PID;
	fb1stORderFilter	: FB_1stOrderFilter;
END_VAR
VAR_INPUT
	Enable			: BOOL;
	Reset			: BOOL;
	TskCycleTime	: TIME;
	CtrlCycleTime	: TIME;
	Invers			: BOOL;
	SP_INT			: REAL;
	SP_HLM			: REAL;
	SP_LLM			: REAL;
	SP_ROC			: REAL;
	PV_IN			: REAL;
	PV_TMLAG		: REAL;
	DEADBAND		: REAL;
	fI_InnerWindow	: REAL;
	ManValue		: REAL;
	Man_On			: BOOL;
	Kp				: REAL;
	Tn				: REAL;
	Tv				: REAL;
	Td				: REAL;
	Output_Min		: REAL;
	Output_Max		: REAL;
	LMN_ROC_UP		: REAL;
	LMN_ROC_DOWN	: REAL;
	LMN_HLM			: REAL;
	LMN_LLM			: REAL;
END_VAR
VAR_OUTPUT
	LMN				: REAL;
END_VAR

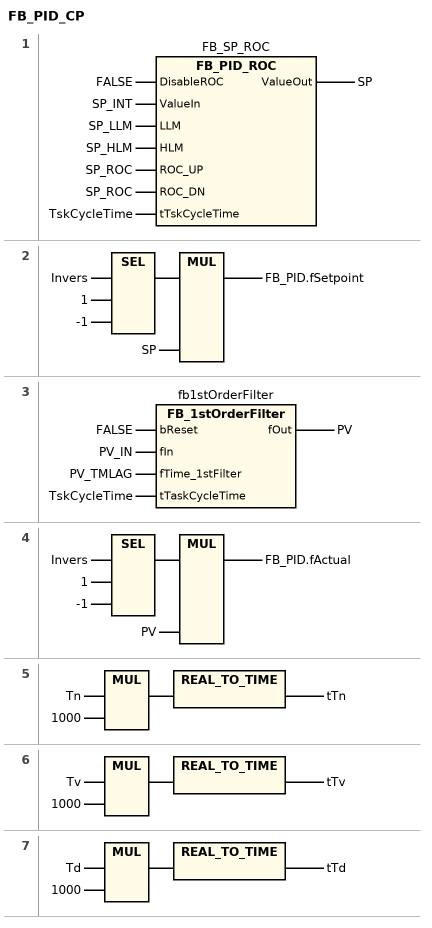
// NETWORK 1
FB_SP_ROC(
    DisableROC := FALSE,
    ValueIn := SP_INT,
    LLM := SP_LLM,
    HLM := SP_HLM,
    ROC_UP := SP_ROC,
    ROC_DN := SP_ROC,
    tTskCycleTime := TskCycleTime); // FB_PID_ROC
SP := FB_SP_ROC.ValueOut;

// NETWORK 2
FB_PID.fSetpoint := SEL(Invers, 1, -1) * SP;

// NETWORK 3
fb1stOrderFilter(bReset := FALSE, fIn := PV_IN, fTime_1stFilter := PV_TMLAG, tTaskCycleTime := TskCycleTime); // FB_1stOrderFilter
PV := fb1stOrderFilter.fOut;

// NETWORK 4
FB_PID.fActual := SEL(Invers, 1, -1) * PV;

// NETWORK 5
tTn := REAL_TO_TIME(Tn * 1000);

// NETWORK 6
tTv := REAL_TO_TIME(Tv * 1000);

// NETWORK 7
tTd := REAL_TO_TIME(Td * 1000);

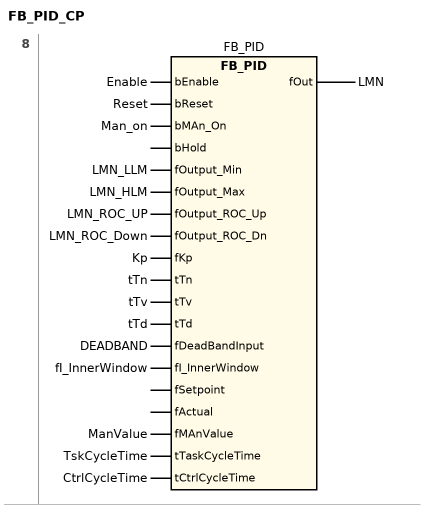
// NETWORK 8
FB_PID(
    bEnable := Enable,
    bReset := Reset,
    bMAn_On := Man_on,
    fOutput_Min := LMN_LLM,
    fOutput_Max := LMN_HLM,
    fOutput_ROC_Up := LMN_ROC_UP,
    fOutput_ROC_Dn := LMN_ROC_Down,
    fKp := Kp,
    tTn := tTn,
    tTv := tTv,
    tTd := tTd,
    fDeadBandInput := DEADBAND,
    fI_InnerWindow := fI_InnerWindow,
    fMAnValue := ManValue,
    tTaskCycleTime := TskCycleTime,
    tCtrlCycleTime := CtrlCycleTime);
LMN := FB_PID.fOut;

END_FUNCTION_BLOCK

// ---- POUs/Standard/HeatingZone/PID/FB_PID_ROC.TcPOU
FUNCTION_BLOCK FB_PID_ROC
VAR_INPUT
	DisableROC			: BOOL;
	ValueIn				: REAL;
	LLM					: REAL; (* Setpoint low limit	*)
	HLM					: REAL; (* Setpoint high limit	*)
	ROC_UP				: REAL;
	ROC_DN				: REAL;
	tTskCycleTime		: TIME;
END_VAR
VAR_OUTPUT
	ValueOut			: REAL;
END_VAR
VAR
	OldValueIN			: REAL;
	ROC_UpLimit			: BOOL;
	ROC_DownLimit			: BOOL;
	CycleTimeSeconds	: REAL;
	ROC_UP_PerCycle		: REAL;
	ROC_DN_PerCycle		: REAL;
END_VAR
VAR // added by the converter: edge detectors and wires of the graphical bodies
    _w1, _w2 : BOOL;
END_VAR

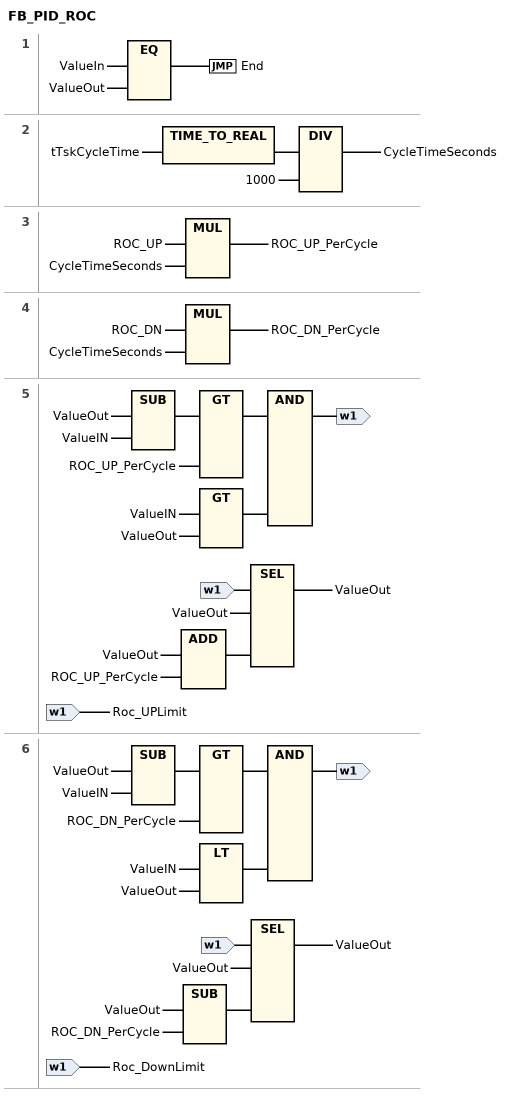
// NETWORK 1
IF ValueIn = ValueOut THEN JMP End; END_IF

// NETWORK 2
CycleTimeSeconds := TIME_TO_REAL(tTskCycleTime) / 1000;

// NETWORK 3
ROC_UP_PerCycle := ROC_UP * CycleTimeSeconds;

// NETWORK 4
ROC_DN_PerCycle := ROC_DN * CycleTimeSeconds;

// NETWORK 5
_w1 := ValueOut - ValueIN > ROC_UP_PerCycle AND ValueIN > ValueOut;
ValueOut := SEL(_w1, ValueOut, ValueOut + ROC_UP_PerCycle);
Roc_UPLimit := _w1;

// NETWORK 6
_w2 := ValueOut - ValueIN > ROC_DN_PerCycle AND ValueIN < ValueOut;
ValueOut := SEL(_w2, ValueOut, ValueOut - ROC_DN_PerCycle);
Roc_DownLimit := _w2;

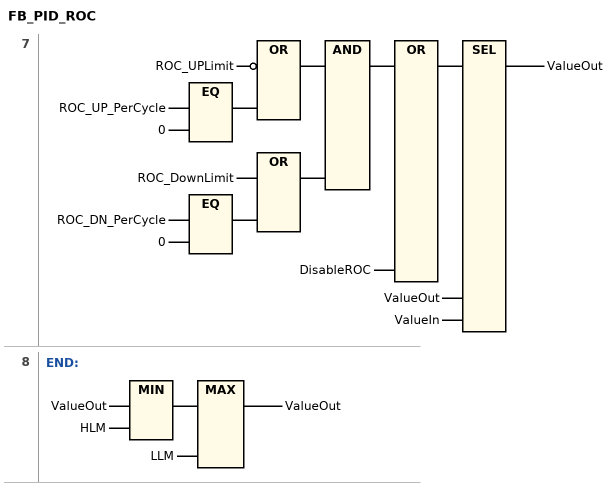
// NETWORK 7
ValueOut := SEL((NOT ROC_UPLimit OR ROC_UP_PerCycle = 0) AND (ROC_DownLimit OR ROC_DN_PerCycle = 0) OR DisableROC, ValueOut, ValueIn);

// NETWORK 8
END:
ValueOut := MAX(MIN(ValueOut, HLM), LLM);

END_FUNCTION_BLOCK

// ---- POUs/Standard/HeatingZone/PID/FB_PID.TcPOU
FUNCTION_BLOCK FB_PID
VAR
	bSync			: BOOL;					(* Synchronize controller							*)
	bSyncSR			: RS;					(* Set reset synchronize controller					*)
	bSyncMaxTime	: TON;					(* Timer for max synchronisation time				*)

	bHoldLocal		: BOOL;					(* Internal hold bit								*)

	eMode			: E_CTRL_MODE;			(* Controller mode									*)
	eState			: E_CTRL_STATE;			(* Controller mode: passive, activ, check, error 	*)

	stParams	: ST_CTRL_PID_EXT_PARAMS;	(* controller External PID parameters				*)

	PID_EXT		: FB_CTRL_PID_EXT;			(* PID controller									*)
	PID_ROC		: FB_PID_ROC;				(* PID rate of change								*)

	bMaxLimitReached	: BOOL := FALSE;	(* Minimum limiting active ? [TRUE/FALSE] -> ARW 	*)
	bMinLimitReached	: BOOL := FALSE;	(* Maximum limiting active ? [TRUE/FALSE] -> ARW 	*)
	bARWActive			: BOOL := FALSE;	(* ARW actice ? [TRUE/FALSE] -> freeze I-part		*)

	ManualFTRIG			: F_TRIG;			(* Trigger for manual mode							*)

	(* auxiliary outputs *)
	fCtrlDerivation		: REAL; 			(* Controller command derivation dy/dt				 *)
	ROCIN				: REAL;				(* Value rate of change input						*)


	(* error outputs *)
	bError				: BOOL;					(* error flag 					*)
	eErrorId			: E_CTRL_ERRORCODES;	(* error code 					*)
	PID_fOut			: REAL;					(* error pid value output		*)
	fOut_Old			: REAL;					(* error value old output value	*)
END_VAR

VAR_INPUT
	bEnable				: BOOL;	(* controller enabled 				*)
	bReset				: BOOL;	(* reset controller 				*)
	bMAn_On				: BOOL;	(* controller in manual				*)
	bHold				: BOOL;	(* hold values						*)
	fOutput_Min			: REAL;	(* minimum value output				*)
	fOutput_Max			: REAL;	(* maximum value output				*)
	fOutput_ROC_Up		: REAL; (* Rate of change value output up	*)
	fOutput_ROC_Dn		: REAL; (* Rate of change value output down	*)
	fKp					: REAL;	(* Proportional value				*)
	tTn					: TIME;	(* Timer Tn time					*)
	tTv					: TIME;	(* Timer Tv time					*)
	tTd					: TIME;	(* Timer Td time					*)
	fDeadBandInput		: REAL;	(* input value deadband				*)
	fI_InnerWindow		: REAL;	(* value inner window				*)
	fSetpoint			: REAL;	(* setpoint value					*)
	fActual				: REAL;	(* actual value						*)
	fMAnValue			: REAL;	(* manual value						*)

	tTaskCycleTime		: TIME;	(* task cycle time					*)
	tCtrlCycleTime		: TIME;	(* control cycle time				*)

END_VAR

VAR_OUTPUT
	fOut				: REAL;	(* output value						*)
END_VAR

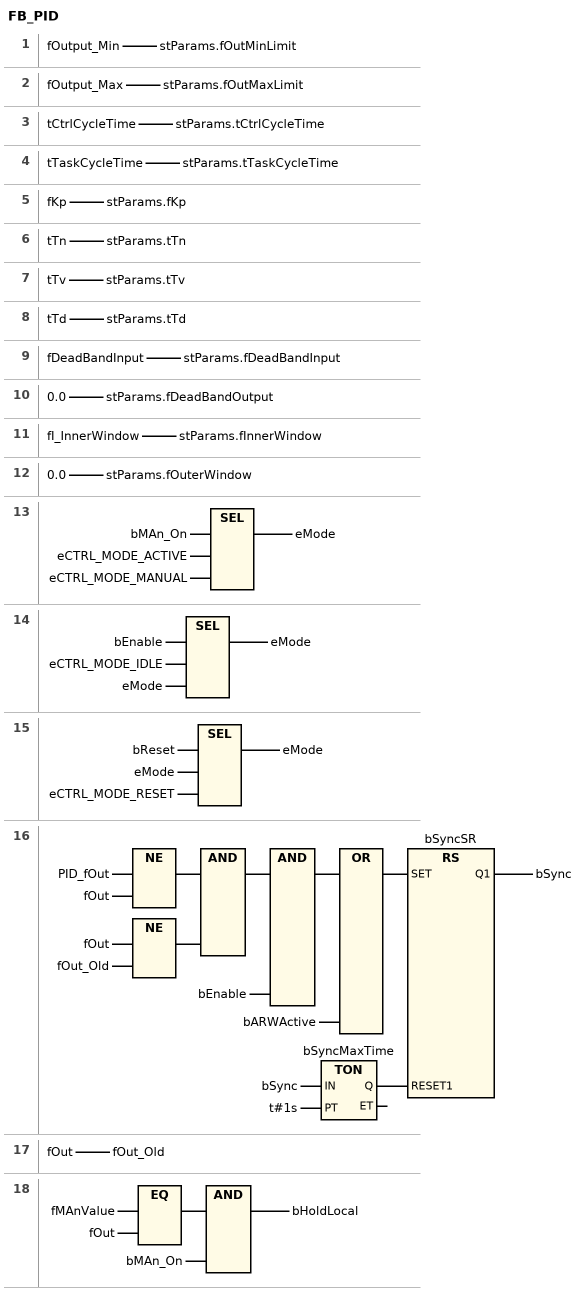
// NETWORK 1
stParams.fOutMinLimit := fOutput_Min;

// NETWORK 2
stParams.fOutMaxLimit := fOutput_Max;

// NETWORK 3
stParams.tCtrlCycleTime := tCtrlCycleTime;

// NETWORK 4
stParams.tTaskCycleTime := tTaskCycleTime;

// NETWORK 5
stParams.fKp := fKp;

// NETWORK 6
stParams.tTn := tTn;

// NETWORK 7
stParams.tTv := tTv;

// NETWORK 8
stParams.tTd := tTd;

// NETWORK 9
stParams.fDeadBandInput := fDeadBandInput;

// NETWORK 10
stParams.fDeadBandOutput := 0.0;

// NETWORK 11
stParams.fInnerWindow := fI_InnerWindow;

// NETWORK 12
stParams.fOuterWindow := 0.0;

// NETWORK 13
eMode := SEL(bMAn_On, eCTRL_MODE_ACTIVE, eCTRL_MODE_MANUAL);

// NETWORK 14
eMode := SEL(bEnable, eCTRL_MODE_IDLE, eMode);

// NETWORK 15
eMode := SEL(bReset, eMode, eCTRL_MODE_RESET);

// NETWORK 16
bSyncMaxTime(IN := bSync, PT := t#1s); // TON
bSyncSR(SET := (PID_fOut <> fOut AND fOut <> fOut_Old) AND bEnable OR bARWActive, RESET1 := bSyncMaxTime.Q); // RS
bSync := bSyncSR.Q1;

// NETWORK 17
fOut_Old := fOut;

// NETWORK 18
bHoldLocal := fMAnValue = fOut AND bMAn_On;

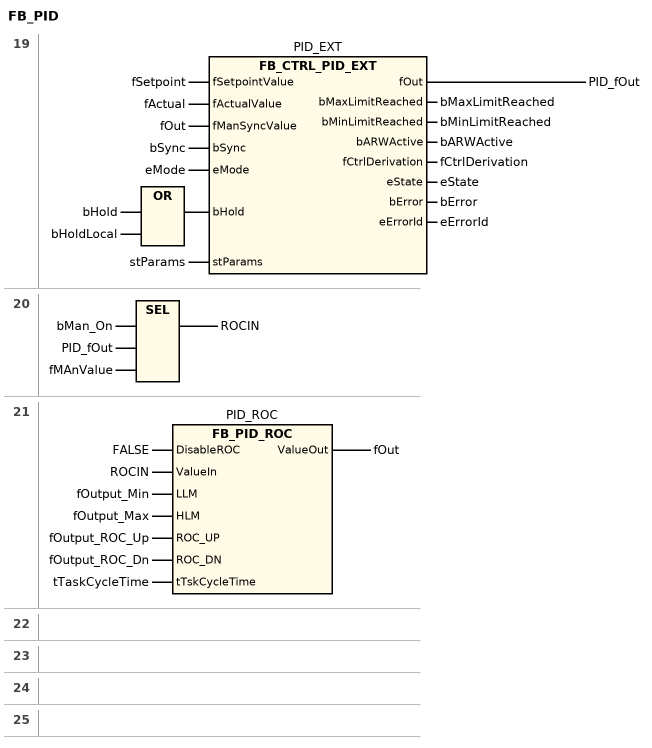
// NETWORK 19
PID_EXT(
    fSetpointValue := fSetpoint,
    fActualValue := fActual,
    fManSyncValue := fOut,
    bSync := bSync,
    eMode := eMode,
    bHold := bHold OR bHoldLocal,
    stParams := stParams,
    bMaxLimitReached => bMaxLimitReached,
    bMinLimitReached => bMinLimitReached,
    bARWActive => bARWActive,
    fCtrlDerivation => fCtrlDerivation,
    eState => eState,
    bError => bError,
    eErrorId => eErrorId); // FB_CTRL_PID_EXT
PID_fOut := PID_EXT.fOut;

// NETWORK 20
ROCIN := SEL(bMan_On, PID_fOut, fMAnValue);

// NETWORK 21
PID_ROC(
    DisableROC := FALSE,
    ValueIn := ROCIN,
    LLM := fOutput_Min,
    HLM := fOutput_Max,
    ROC_UP := fOutput_ROC_Up,
    ROC_DN := fOutput_ROC_Dn,
    tTskCycleTime := tTaskCycleTime); // FB_PID_ROC
fOut := PID_ROC.ValueOut;

// NETWORK 22

// NETWORK 23

// NETWORK 24

// NETWORK 25

END_FUNCTION_BLOCK

// ---- POUs/Standard/HeatingZone/PID/FB_1stOrderFilter.TcPOU
FUNCTION_BLOCK FB_1stOrderFilter
VAR_INPUT
	bReset			: BOOL; (*Reset 1st order filter*)
	fIn				: REAL;	(*Input value*)
	fTime_1stFilter	: REAL;	(*First order filter time in seconds*)
	tTaskCycleTime	: TIME;

	//FB_CTRL_PT1: FB_CTRL_PT1;
END_VAR
VAR_OUTPUT
	fOut			: REAL; (*Output value 2nd Order filtered*)
END_VAR
VAR_IN_OUT

END_VAR

VAR
	bHold						: BOOL;
	bSync						: BOOL;
	bFilterActive				: BOOL;

	eMode						: E_CTRL_MODE;
	eState						: E_CTRL_STATE;

	FB_CTRL_PT1					: FB_CTRL_PT1;
	stCTRL_PT1_PARAMS			: ST_CTRL_PT1_PARAMS;
END_VAR

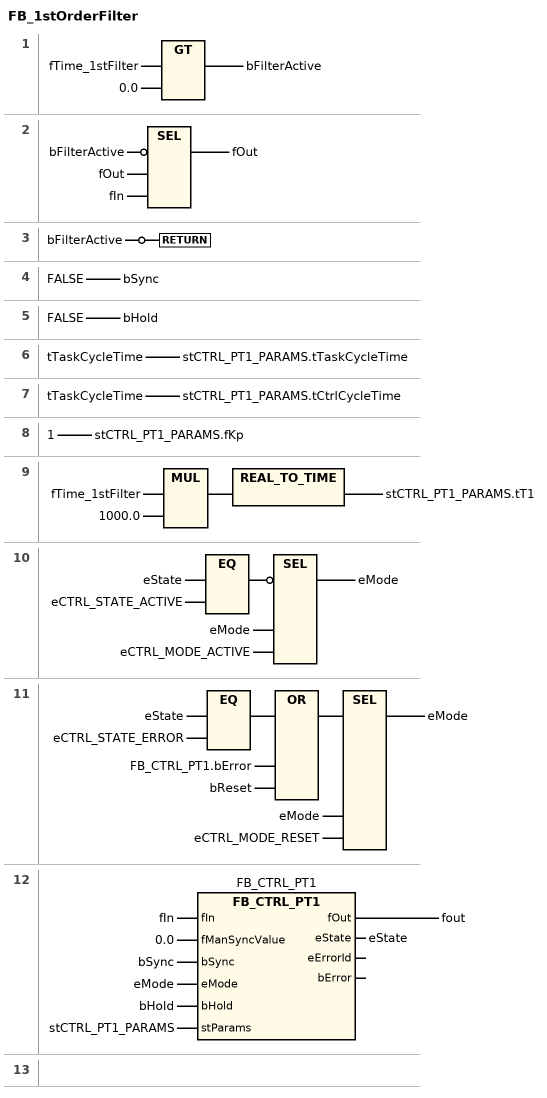
// NETWORK 1
bFilterActive := fTime_1stFilter > 0.0;

// NETWORK 2
fOut := SEL(NOT bFilterActive, fOut, fIn);

// NETWORK 3
IF NOT bFilterActive THEN RETURN; END_IF

// NETWORK 4
bSync := FALSE;

// NETWORK 5
bHold := FALSE;

// NETWORK 6
stCTRL_PT1_PARAMS.tTaskCycleTime := tTaskCycleTime;

// NETWORK 7
stCTRL_PT1_PARAMS.tCtrlCycleTime := tTaskCycleTime;

// NETWORK 8
stCTRL_PT1_PARAMS.fKp := 1;

// NETWORK 9
stCTRL_PT1_PARAMS.tT1 := REAL_TO_TIME(fTime_1stFilter * 1000.0);

// NETWORK 10
eMode := SEL(NOT (eState = eCTRL_STATE_ACTIVE), eMode, eCTRL_MODE_ACTIVE);

// NETWORK 11
eMode := SEL(eState = eCTRL_STATE_ERROR OR FB_CTRL_PT1.bError OR bReset, eMode, eCTRL_MODE_RESET);

// NETWORK 12
FB_CTRL_PT1(
    fIn := fIn,
    fManSyncValue := 0.0,
    bSync := bSync,
    eMode := eMode,
    bHold := bHold,
    stParams := stCTRL_PT1_PARAMS,
    eState => eState);
fout := FB_CTRL_PT1.fOut;

// NETWORK 13

END_FUNCTION_BLOCK

// ---- POUs/Standard/Analog/FB_AnalogInPT100.TcPOU
FUNCTION_BLOCK FB_AnalogInPT100
VAR_INPUT
END_VAR
VAR_OUTPUT
	EngTempOut			: REAL; (*Output in engineering units*)
	Error				: BOOL;
	Wirebreak			: BOOL;
END_VAR
VAR
	RawInput 			AT %I*: INT;
	Status				AT %I*: WORD;
	Underrange			: BOOL;
	Overrange			: BOOL;


END_VAR

Underrange:= Status.0;
Overrange:= Status.1;
Error:= Status.4 OR UnderRange OR Overrange;
Wirebreak := Status.4;


EngTempOut:= INT_TO_REAL(RawInput)/10;

END_FUNCTION_BLOCK

// ---- POUs/HMI.TcPOU
PROGRAM HMI
VAR_OUTPUT
	mxError		:BOOL; (*Error present*)
END_VAR

VAR
(*HMI Vars*)
	AlarmWord1 :DINT;	(* General *)
	AlarmWord2 :DINT;	(* General *)
	AlarmWord3 :DINT;	(* TopMold A *)
	AlarmWord4 :DINT;	(* TopMold A *)
	AlarmWord5 :DINT;	(* TopMold B *)
	AlarmWord6 :DINT;	(* TopMold B *)
	AlarmWord7 :DINT;	(* BottomMold A *)	
	AlarmWord8 :DINT;	(* BottomMold A *)
	AlarmWord9 :DINT;	(* BottomMold A *)
	AlarmWord10 :DINT;	(* BottomMold A *)
	AlarmWord11 :DINT;	(* BottomMold B *)
	AlarmWord12 :DINT;	(* BottomMold B *)
	AlarmWord13 :DINT;	(* BottomMold B *)
	AlarmWord14 :DINT;	(* BottomMold B *)
	AlarmWord15 :DINT;	(* TransferMold *)
	AlarmWord16 :DINT;	(* TransferMold *)
	AlarmWord17 :DINT;	(* ProductForming *)
	AlarmWord18 :DINT;	(* ProductForming *)
	AlarmWord19 :DINT;	(* ProductForming *)
	AlarmWord20 :DINT;	(* ProductForming *)


	sUserName	: STRING	:= 'NONE';
	miUserLevel	: INT		:= 0;

	mxReset		: BOOL;
	T_HmiReset	: TON;
	T_LogOut	: TON;

	mxAutoMode: BOOL;
	
